C01819=1049.631,44.124,-78.703,170.591,33.560,156.310
C01820=1049.638,44.373,-78.720,170.592,33.562,156.310
C01821=1049.643,44.623,-78.737,170.594,33.564,156.311
C01822=1049.650,44.872,-78.754,170.596,33.566,156.311
C01823=1049.656,45.158,-78.774,170.597,33.568,156.311
C01824=1049.664,45.444,-78.793,170.599,33.571,156.312
C01825=1049.671,45.731,-78.812,170.601,33.573,156.312
C01826=1049.678,46.017,-78.832,170.603,33.575,156.312
C01827=1049.684,46.266,-78.848,170.605,33.577,156.313
C01828=1049.690,46.516,-78.866,170.606,33.579,156.313
C01829=1049.696,46.765,-78.883,170.608,33.581,156.313
C01830=1049.702,47.014,-78.900,170.610,33.583,156.314
C01831=1049.709,47.263,-78.917,170.611,33.585,156.314
C01832=1049.714,47.513,-78.934,170.613,33.587,156.314
C01833=1049.721,47.762,-78.951,170.615,33.589,156.315
C01834=1049.727,48.012,-78.967,170.617,33.590,156.315
C01835=1049.732,48.261,-78.985,170.619,33.592,156.315
C01836=1049.739,48.510,-79.002,170.620,33.594,156.316
C01837=1049.745,48.759,-79.018,170.622,33.596,156.316
C01838=1049.751,49.008,-79.036,170.624,33.598,156.316
C01839=1049.757,49.258,-79.053,170.625,33.600,156.316
C01840=1049.763,49.507,-79.070,170.627,33.602,156.317
C01841=1049.770,49.757,-79.088,170.629,33.604,156.317
C01842=1049.775,50.006,-79.104,170.630,33.606,156.317
C01843=1049.781,50.255,-79.121,170.632,33.608,156.318
C01844=1049.788,50.505,-79.139,170.634,33.610,156.318
C01845=1049.794,50.754,-79.155,170.635,33.612,156.318
C01846=1049.800,51.004,-79.173,170.637,33.614,156.319
C01847=1049.806,51.253,-79.190,170.638,33.616,156.319
C01848=1049.813,51.503,-79.207,170.640,33.618,156.319
C01849=1049.818,51.752,-79.224,170.642,33.620,156.320
C01850=1049.825,52.001,-79.241,170.643,33.622,156.320
C01851=1049.831,52.250,-79.258,170.645,33.624,156.320
C01852=1049.837,52.499,-79.275,170.647,33.626,156.321
C01853=1049.843,52.749,-79.293,170.648,33.628,156.321
C01854=1049.850,52.998,-79.310,170.650,33.630,156.321
C01855=1049.856,53.247,-79.327,170.652,33.632,156.322
C01856=1049.862,53.497,-79.344,170.653,33.633,156.322
C01857=1049.868,53.746,-79.362,170.655,33.635,156.322
C01858=1049.874,53.995,-79.379,170.656,33.637,156.322
C01859=1049.881,54.245,-79.396,170.658,33.639,156.323
C01860=1049.886,54.494,-79.413,170.660,33.641,156.323
C01861=1049.893,54.744,-79.430,170.661,33.643,156.323
C01862=1049.899,54.992,-79.447,170.663,33.645,156.324
C01863=1049.905,55.242,-79.465,170.665,33.647,156.324
C01864=1049.912,55.491,-79.482,170.666,33.649,156.324
C01865=1049.918,55.741,-79.499,170.668,33.651,156.325
C01866=1049.924,55.990,-79.516,170.670,33.653,156.325
C01867=1049.931,56.239,-79.534,170.671,33.655,156.325
C01868=1049.936,56.488,-79.551,170.673,33.657,156.326
C01869=1049.943,56.738,-79.568,170.674,33.659,156.326
C01870=1049.949,56.988,-79.586,170.676,33.660,156.326
C01871=1049.955,57.236,-79.603,170.678,33.662,156.326
C01872=1049.962,57.486,-79.620,170.679,33.664,156.327
C01873=1049.967,57.735,-79.638,170.681,33.666,156.327
C01874=1049.974,57.985,-79.655,170.684,33.668,156.327
C01875=1049.980,58.234,-79.672,170.685,33.670,156.328
C01876=1049.987,58.483,-79.690,170.687,33.672,156.328
C01877=1049.994,58.733,-79.707,170.689,33.674,156.328
C01878=1049.999,58.982,-79.725,170.690,33.676,156.329
C01879=1050.006,59.231,-79.742,170.692,33.678,156.329
C01880=1050.011,59.480,-79.760,170.693,33.680,156.329
C01881=1050.018,59.730,-79.777,170.695,33.682,156.330
C01882=1050.024,59.979,-79.795,170.697,33.683,156.330
C01883=1050.031,60.228,-79.812,170.698,33.685,156.330
C01884=1050.038,60.478,-79.829,170.700,33.687,156.330
C01885=1050.043,60.727,-79.847,170.702,33.689,156.331
C01886=1050.050,60.976,-79.864,170.703,33.691,156.331
C01887=1050.057,61.262,-79.884,170.705,33.693,156.331
C01888=1050.064,61.548,-79.904,170.707,33.696,156.332
C01889=1050.071,61.834,-79.924,170.709,33.698,156.332
C01890=1050.079,62.120,-79.943,170.711,33.700,156.332
C01891=1050.085,62.369,-79.961,170.712,33.702,156.333
C01892=1050.091,62.619,-79.979,170.714,33.704,156.333
C01893=1050.097,62.868,-79.996,170.716,33.706,156.333
C01894=1050.104,63.117,-80.014,170.717,33.708,156.334
C01895=1050.110,63.366,-80.032,170.719,33.710,156.334
C01896=1050.117,63.615,-80.049,170.721,33.712,156.334
C01897=1050.123,63.865,-80.067,170.722,33.713,156.335
C01898=1050.130,64.114,-80.084,170.724,33.715,156.335
C01899=1050.135,64.363,-80.102,170.726,33.717,156.335
C01900=1050.142,64.613,-80.119,170.727,33.719,156.336
C01901=1050.148,64.862,-80.137,170.729,33.721,156.336
C01902=1050.154,65.111,-80.155,170.730,33.723,156.336
C01903=1050.160,65.361,-80.173,170.732,33.725,156.337
C01904=1050.167,65.610,-80.191,170.734,33.727,156.337
C01905=1050.172,65.859,-80.208,170.735,33.729,156.337
C01906=1050.178,66.109,-80.226,170.737,33.731,156.337
C01907=1050.185,66.358,-80.244,170.739,33.733,156.338
C01908=1050.191,66.607,-80.261,170.741,33.734,156.338
C01909=1050.197,66.856,-80.280,170.743,33.736,156.338
C01910=1050.204,67.106,-80.297,170.744,33.738,156.339
C01911=1050.210,67.355,-80.315,170.746,33.741,156.339
C01912=1050.216,67.605,-80.333,170.748,33.743,156.340
C01913=1050.222,67.854,-80.351,170.749,33.745,156.340
C01914=1050.228,68.102,-80.368,170.751,33.747,156.340
C01915=1050.235,68.352,-80.386,170.753,33.749,156.340
C01916=1050.241,68.602,-80.404,170.754,33.751,156.341
C01917=1050.247,68.850,-80.422,170.756,33.753,156.341
C01918=1050.253,69.100,-80.440,170.757,33.755,156.341
C01919=1050.259,69.350,-80.458,170.759,33.757,156.342
C01920=1050.265,69.599,-80.475,170.761,33.759,156.342
C01921=1050.271,69.848,-80.494,170.762,33.761,156.342
C01922=1050.278,70.097,-80.512,170.764,33.763,156.343
C01923=1050.283,70.346,-80.529,170.766,33.764,156.343
C01924=1050.290,70.596,-80.548,170.767,33.766,156.343
C01925=1050.296,70.845,-80.565,170.769,33.768,156.344
C01926=1050.302,71.094,-80.583,170.770,33.770,156.344
C01927=1050.308,71.343,-80.602,170.772,33.772,156.344
C01928=1050.314,71.593,-80.620,170.774,33.774,156.345
C01929=1050.321,71.843,-80.638,170.775,33.776,156.345
C01930=1050.326,72.091,-80.656,170.777,33.778,156.345
C01931=1050.332,72.341,-80.674,170.779,33.780,156.346
C01932=1050.339,72.590,-80.692,170.780,33.783,156.346
C01933=1050.345,72.840,-80.710,170.782,33.785,156.346
C01934=1050.351,73.088,-80.727,170.783,33.787,156.347
C01935=1050.358,73.338,-80.746,170.786,33.789,156.347
C01936=1050.364,73.587,-80.764,170.788,33.791,156.347
C01937=1050.370,73.836,-80.782,170.789,33.792,156.348
C01938=1050.376,74.085,-80.800,170.791,33.794,156.348
C01939=1050.382,74.335,-80.819,170.792,33.796,156.348
C01940=1050.388,74.584,-80.837,170.794,33.798,156.349
C01941=1050.395,74.833,-80.855,170.796,33.800,156.349
C01942=1050.400,75.082,-80.873,170.797,33.802,156.349
C01943=1050.407,75.332,-80.892,170.799,33.804,156.350
C01944=1050.413,75.581,-80.909,170.801,33.806,156.350
C01945=1050.419,75.830,-80.928,170.802,33.808,156.350
C01946=1050.425,76.079,-80.946,170.804,33.810,156.351
C01947=1050.431,76.329,-80.964,170.805,33.812,156.351
C01948=1050.437,76.578,-80.982,170.807,33.814,156.351
C01949=1050.444,76.827,-81.000,170.809,33.816,156.352
C01950=1050.451,77.077,-81.018,170.810,33.819,156.352
C01951=1050.457,77.363,-81.040,170.812,33.821,156.352
C01952=1050.464,77.648,-81.060,170.814,33.823,156.353
C01953=1050.471,77.933,-81.081,170.816,33.825,156.353
C01954=1050.479,78.219,-81.102,170.818,33.828,156.353
C01955=1050.484,78.468,-81.120,170.819,33.830,156.354
C01956=1050.491,78.718,-81.139,170.821,33.832,156.354
C01957=1050.496,78.967,-81.158,170.823,33.834,156.354
C01958=1050.503,79.217,-81.176,170.824,33.835,156.355
C01959=1050.509,79.466,-81.195,170.827,33.837,156.355
C01960=1050.515,79.714,-81.213,170.828,33.839,156.355
C01961=1050.521,79.964,-81.231,170.830,33.842,156.356
C01962=1050.527,80.213,-81.249,170.832,33.844,156.356
C01963=1050.533,80.463,-81.269,170.833,33.846,156.357
C01964=1050.539,80.712,-81.287,170.835,33.848,156.357
C01965=1050.545,80.961,-81.305,170.837,33.850,156.357
C01966=1050.551,81.210,-81.323,170.838,33.852,156.357
C01967=1050.558,81.460,-81.341,170.840,33.854,156.358
C01968=1050.563,81.709,-81.361,170.841,33.856,156.358
C01969=1050.570,81.958,-81.379,170.843,33.858,156.359
C01970=1050.576,82.207,-81.398,170.845,33.860,156.359
C01971=1050.582,82.456,-81.416,170.846,33.862,156.359
C01972=1050.588,82.705,-81.434,170.848,33.864,156.360
C01973=1050.594,82.955,-81.453,170.849,33.866,156.360
C01974=1050.600,83.204,-81.472,170.851,33.868,156.360
C01975=1050.606,83.454,-81.490,170.853,33.871,156.361
C01976=1050.613,83.703,-81.509,170.854,33.872,156.361
C01977=1050.618,83.952,-81.528,170.856,33.874,156.361
C01978=1050.624,84.201,-81.546,170.858,33.876,156.362
C01979=1050.630,84.450,-81.564,170.859,33.878,156.362
C01980=1050.637,84.700,-81.583,170.861,33.880,156.362
C01981=1050.643,84.949,-81.601,170.863,33.882,156.363
C01982=1050.649,85.198,-81.621,170.865,33.884,156.363
C01983=1050.655,85.447,-81.639,170.867,33.887,156.363
C01984=1050.662,85.696,-81.658,170.868,33.889,156.364
C01985=1050.668,85.946,-81.676,170.870,33.891,156.364
C01986=1050.674,86.196,-81.695,170.872,33.893,156.364
C01987=1050.680,86.445,-81.714,170.873,33.895,156.365
C01988=1050.686,86.693,-81.732,170.875,33.896,156.365
C01989=1050.692,86.942,-81.751,170.876,33.898,156.365
C01990=1050.699,87.191,-81.769,170.878,33.900,156.366
C01991=1050.704,87.441,-81.789,170.880,33.902,156.366
C01992=1050.711,87.690,-81.807,170.881,33.905,156.366
C01993=1050.717,87.940,-81.825,170.883,33.907,156.367
C01994=1050.723,88.189,-81.844,170.885,33.909,156.367
C01995=1050.729,88.438,-81.863,170.886,33.911,156.367
C01996=1050.735,88.687,-81.882,170.888,33.913,156.368
C01997=1050.742,88.936,-81.900,170.890,33.915,156.368
C01998=1050.748,89.186,-81.919,170.891,33.917,156.368
C01999=1050.754,89.435,-81.938,170.893,33.919,156.369
C02000=1050.760,89.684,-81.957,170.894,33.920,156.369
C02001=1050.767,89.933,-81.976,170.896,33.922,156.369
C02002=1050.772,90.183,-81.995,170.898,33.924,156.370
C02003=1050.779,90.432,-82.013,170.900,33.926,156.370
C02004=1050.785,90.681,-82.032,170.902,33.929,156.370
C02005=1050.791,90.930,-82.051,170.904,33.931,156.371
C02006=1050.797,91.179,-82.070,170.905,33.933,156.371
C02007=1050.803,91.429,-82.089,170.907,33.935,156.371
C02008=1050.810,91.678,-82.108,170.908,33.937,156.372
C02009=1050.815,91.927,-82.127,170.910,33.939,156.372
C02010=1050.822,92.177,-82.146,170.912,33.941,156.372
C02011=1050.827,92.426,-82.165,170.913,33.943,156.373
C02012=1050.834,92.675,-82.184,170.915,33.945,156.373
C02013=1050.840,92.924,-82.204,170.917,33.948,156.374
C02014=1050.846,93.173,-82.222,170.918,33.950,156.374
C02015=1050.853,93.459,-82.244,170.920,33.952,156.374
C02016=1050.860,93.744,-82.266,170.922,33.954,156.375
C02017=1050.867,94.030,-82.287,170.924,33.957,156.375
C02018=1050.874,94.315,-82.309,170.926,33.959,156.375
C02019=1050.879,94.564,-82.328,170.927,33.961,156.376
C02020=1050.886,94.814,-82.347,170.929,33.963,156.376
C02021=1050.891,95.063,-82.366,170.932,33.965,156.376
C02022=1050.897,95.312,-82.386,170.933,33.967,156.377
C02023=1050.904,95.562,-82.405,170.935,33.969,156.377
C02024=1050.910,95.811,-82.424,170.937,33.972,156.378
C02025=1050.916,96.060,-82.443,170.938,33.973,156.378
C02026=1050.922,96.310,-82.462,170.940,33.975,156.378
C02027=1050.929,96.558,-82.482,170.941,33.977,156.379
C02028=1050.935,96.808,-82.501,170.943,33.979,156.379
C02029=1050.941,97.057,-82.520,170.945,33.981,156.379
C02030=1050.947,97.306,-82.539,170.946,33.984,156.380
C02031=1050.953,97.555,-82.558,170.948,33.986,156.380
C02032=1050.959,97.804,-82.577,170.950,33.988,156.380
C02033=1050.965,98.053,-82.597,170.951,33.990,156.381
C02034=1050.971,98.303,-82.615,170.953,33.992,156.381
C02035=1050.977,98.552,-82.635,170.955,33.994,156.381
C02036=1050.984,98.801,-82.654,170.956,33.996,156.382
C02037=1050.989,99.050,-82.673,170.958,33.998,156.382
C02038=1050.996,99.300,-82.692,170.960,34.000,156.382
C02039=1051.002,99.549,-82.712,170.962,34.002,156.383
C02040=1051.009,99.798,-82.731,170.964,34.004,156.383
C02041=1051.014,100.047,-82.750,170.966,34.006,156.383
C02042=1051.020,100.296,-82.770,170.967,34.008,156.384
C02043=1051.027,100.545,-82.789,170.969,34.010,156.384
C02044=1051.033,100.795,-82.808,170.970,34.012,156.384
C02045=1051.039,101.043,-82.828,170.972,34.014,156.385
C02046=1051.045,101.292,-82.847,170.974,34.016,156.385
C02047=1051.051,101.542,-82.866,170.975,34.019,156.386
C02048=1051.057,101.791,-82.886,170.977,34.021,156.386
C02049=1051.063,102.041,-82.905,170.979,34.023,156.386
C02050=1051.069,102.290,-82.925,170.980,34.024,156.387
C02051=1051.075,102.539,-82.944,170.982,34.027,156.387
C02052=1051.081,102.788,-82.964,170.984,34.029,156.387
C02053=1051.087,103.037,-82.983,170.985,34.031,156.388
C02054=1051.093,103.286,-83.003,170.987,34.033,156.388
C02055=1051.099,103.535,-83.022,170.989,34.035,156.388
C02056=1051.105,103.784,-83.042,170.991,34.037,156.389
C02057=1051.111,104.033,-83.061,170.993,34.039,156.389
C02058=1051.117,104.283,-83.081,170.995,34.042,156.389
C02059=1051.123,104.532,-83.101,170.996,34.044,156.390
C02060=1051.129,104.782,-83.120,170.998,34.046,156.390
C02061=1051.135,105.030,-83.140,170.999,34.048,156.390
C02062=1051.142,105.279,-83.159,171.001,34.050,156.391
C02063=1051.148,105.528,-83.178,171.003,34.052,156.391
C02064=1051.154,105.777,-83.198,171.004,34.054,156.392
C02065=1051.160,106.027,-83.218,171.006,34.056,156.392
C02066=1051.166,106.276,-83.238,171.008,34.059,156.392
C02067=1051.172,106.526,-83.257,171.009,34.060,156.393
C02068=1051.178,106.774,-83.276,171.011,34.062,156.393
C02069=1051.184,107.023,-83.296,171.013,34.064,156.393
C02070=1051.191,107.273,-83.316,171.014,34.066,156.394
C02071=1051.197,107.522,-83.336,171.016,34.069,156.394
C02072=1051.202,107.771,-83.355,171.019,34.071,156.394
C02073=1051.208,108.020,-83.375,171.020,34.073,156.395
C02074=1051.215,108.269,-83.394,171.022,34.075,156.395
C02075=1051.221,108.519,-83.414,171.024,34.077,156.396
C02076=1051.227,108.767,-83.434,171.025,34.079,156.396
C02077=1051.233,109.017,-83.453,171.027,34.081,156.396
C02078=1051.239,109.266,-83.473,171.029,34.083,156.397
C02079=1051.246,109.551,-83.496,171.031,34.086,156.397
C02080=1051.253,109.837,-83.519,171.033,34.088,156.397
C02081=1051.260,110.123,-83.541,171.035,34.090,156.398
C02082=1051.267,110.408,-83.564,171.036,34.093,156.398
C02083=1051.274,110.658,-83.583,171.038,34.095,156.399
C02084=1051.280,110.906,-83.603,171.040,34.097,156.399
C02085=1051.286,111.155,-83.623,171.041,34.099,156.399
C02086=1051.292,111.405,-83.642,171.043,34.101,156.400
C02087=1051.298,111.654,-83.663,171.045,34.103,156.400
C02088=1051.304,111.903,-83.683,171.048,34.105,156.400
C02089=1051.310,112.152,-83.703,171.049,34.107,156.401
C02090=1051.316,112.401,-83.722,171.051,34.109,156.401
C02091=1051.322,112.651,-83.742,171.053,34.111,156.401
C02092=1051.328,112.900,-83.762,171.054,34.114,156.402
C02093=1051.334,113.148,-83.782,171.056,34.116,156.402
C02094=1051.340,113.397,-83.802,171.058,34.118,156.402
C02095=1051.347,113.647,-83.822,171.059,34.120,156.403
C02096=1051.353,113.896,-83.842,171.061,34.122,156.403
C02097=1051.358,114.145,-83.862,171.063,34.124,156.404
C02098=1051.364,114.394,-83.882,171.064,34.126,156.404
C02099=1051.371,114.644,-83.903,171.066,34.129,156.404
C02100=1051.377,114.892,-83.922,171.068,34.131,156.405
C02101=1051.382,115.142,-83.943,171.069,34.133,156.405
C02102=1051.388,115.390,-83.963,171.072,34.135,156.405
C02103=1051.394,115.641,-83.983,171.074,34.137,156.406
C02104=1051.399,115.890,-84.003,171.075,34.139,156.406
C02105=1051.405,116.138,-84.023,171.077,34.141,156.407
C02106=1051.411,116.387,-84.043,171.079,34.144,156.407
C02107=1051.418,116.637,-84.063,171.080,34.146,156.407
C02108=1051.423,116.886,-84.084,171.082,34.148,156.408
C02109=1051.429,117.135,-84.104,171.084,34.150,156.408
C02110=1051.436,117.384,-84.124,171.085,34.152,156.408
C02111=1051.442,117.633,-84.144,171.087,34.154,156.409
C02112=1051.447,117.882,-84.165,171.089,34.157,156.409
C02113=1051.453,118.131,-84.185,171.090,34.159,156.410
C02114=1051.460,118.381,-84.205,171.092,34.161,156.410
C02115=1051.466,118.629,-84.225,171.094,34.163,156.410
C02116=1051.471,118.878,-84.246,171.096,34.165,156.411
C02117=1051.477,119.128,-84.266,171.098,34.168,156.411
C02118=1051.483,119.377,-84.286,171.100,34.170,156.411
C02119=1051.489,119.626,-84.306,171.102,34.172,156.412
C02120=1051.495,119.875,-84.327,171.103,34.174,156.412
C02121=1051.501,120.124,-84.347,171.105,34.176,156.413
C02122=1051.507,120.373,-84.367,171.107,34.179,156.413
C02123=1051.513,120.623,-84.388,171.108,34.180,156.413
C02124=1051.519,120.871,-84.408,171.110,34.182,156.414
C02125=1051.525,121.120,-84.428,171.112,34.185,156.414
C02126=1051.531,121.370,-84.449,171.113,34.187,156.414
C02127=1051.537,121.619,-84.469,171.115,34.189,156.415
C02128=1051.543,121.867,-84.489,171.117,34.191,156.415
C02129=1051.549,122.117,-84.510,171.119,34.193,156.416
C02130=1051.555,122.366,-84.530,171.121,34.195,156.416
C02131=1051.562,122.615,-84.550,171.123,34.198,156.416
C02132=1051.567,122.864,-84.571,171.125,34.200,156.417
C02133=1051.573,123.113,-84.591,171.126,34.202,156.417
C02134=1051.580,123.362,-84.612,171.128,34.204,156.417
C02135=1051.585,123.611,-84.632,171.130,34.206,156.418
C02136=1051.592,123.861,-84.653,171.132,34.208,156.418
C02137=1051.598,124.110,-84.673,171.133,34.211,156.419
C02138=1051.604,124.358,-84.693,171.135,34.212,156.419
C02139=1051.610,124.608,-84.714,171.137,34.214,156.419
C02140=1051.616,124.857,-84.734,171.138,34.217,156.420
C02141=1051.622,125.106,-84.754,171.140,34.219,156.420
C02142=1051.628,125.355,-84.775,171.142,34.221,156.420
C02143=1051.635,125.641,-84.799,171.145,34.223,156.421
C02144=1051.642,125.926,-84.822,171.147,34.226,156.421
C02145=1051.649,126.211,-84.846,171.149,34.228,156.422
C02146=1051.656,126.497,-84.870,171.151,34.231,156.422
C02147=1051.662,126.746,-84.890,171.153,34.233,156.422
C02148=1051.668,126.995,-84.910,171.154,34.235,156.423
C02149=1051.675,127.244,-84.932,171.156,34.237,156.423
C02150=1051.681,127.493,-84.952,171.158,34.239,156.423
C02151=1051.687,127.743,-84.972,171.160,34.241,156.424
C02152=1051.693,127.991,-84.993,171.161,34.243,156.424
C02153=1051.699,128.241,-85.013,171.163,34.246,156.425
C02154=1051.705,128.490,-85.034,171.165,34.248,156.425
C02155=1051.711,128.739,-85.055,171.167,34.250,156.425
C02156=1051.717,128.988,-85.075,171.169,34.252,156.426
C02157=1051.723,129.237,-85.096,171.171,34.254,156.426
C02158=1051.730,129.486,-85.117,171.173,34.256,156.426
C02159=1051.736,129.735,-85.137,171.175,34.259,156.427
C02160=1051.741,129.984,-85.157,171.176,34.260,156.427
C02161=1051.748,130.233,-85.179,171.178,34.262,156.427
C02162=1051.754,130.482,-85.198,171.180,34.265,156.428
C02163=1051.760,130.731,-85.220,171.182,34.267,156.428
C02164=1051.766,130.980,-85.240,171.183,34.269,156.429
C02165=1051.772,131.230,-85.261,171.185,34.271,156.429
C02166=1051.779,131.479,-85.282,171.187,34.273,156.429
C02167=1051.784,131.728,-85.303,171.189,34.275,156.430
C02168=1051.791,131.977,-85.324,171.191,34.278,156.430
C02169=1051.797,132.226,-85.344,171.193,34.280,156.430
C02170=1051.803,132.475,-85.366,171.195,34.282,156.431
C02171=1051.809,132.724,-85.386,171.197,34.284,156.431
C02172=1051.815,132.973,-85.407,171.198,34.286,156.432
C02173=1051.820,133.222,-85.428,171.200,34.289,156.432
C02174=1051.827,133.471,-85.449,171.202,34.290,156.432
C02175=1051.833,133.720,-85.470,171.204,34.293,156.433
C02176=1051.839,133.969,-85.491,171.205,34.295,156.433
C02177=1051.845,134.218,-85.512,171.207,34.297,156.434
C02178=1051.851,134.467,-85.533,171.209,34.299,156.434
C02179=1051.857,134.717,-85.554,171.211,34.301,156.434
C02180=1051.863,134.965,-85.574,171.213,34.304,156.435
C02181=1051.869,135.215,-85.596,171.215,34.306,156.435
C02182=1051.875,135.463,-85.617,171.217,34.308,156.436
C02183=1051.881,135.713,-85.638,171.219,34.310,156.436
C02184=1051.887,135.961,-85.659,171.221,34.313,156.436
C02185=1051.893,136.210,-85.681,171.222,34.315,156.437
C02186=1051.900,136.460,-85.701,171.224,34.317,156.437
C02187=1051.905,136.708,-85.722,171.226,34.319,156.437
C02188=1051.911,136.958,-85.744,171.228,34.321,156.438
C02189=1051.917,137.206,-85.764,171.229,34.324,156.438
C02190=1051.923,137.456,-85.785,171.231,34.325,156.439
C02191=1051.930,137.705,-85.807,171.233,34.328,156.439
C02192=1051.935,137.954,-85.828,171.236,34.330,156.439
C02193=1051.942,138.203,-85.849,171.238,34.332,156.440
C02194=1051.947,138.451,-85.870,171.239,34.334,156.440
C02195=1051.953,138.700,-85.891,171.241,34.336,156.440
C02196=1051.959,138.950,-85.912,171.243,34.339,156.441
C02197=1051.966,139.199,-85.933,171.245,34.341,156.441
C02198=1051.972,139.448,-85.955,171.246,34.343,156.442
C02199=1051.978,139.697,-85.976,171.248,34.345,156.442
C02200=1051.983,139.946,-85.997,171.250,34.348,156.442
C02201=1051.989,140.195,-86.019,171.252,34.350,156.443
C02202=1051.995,140.444,-86.040,171.254,34.352,156.443
C02203=1052.001,140.693,-86.061,171.256,34.354,156.444
C02204=1052.008,140.942,-86.082,171.258,34.357,156.444
C02205=1052.013,141.191,-86.103,171.260,34.359,156.444
C02206=1052.019,141.440,-86.125,171.262,34.361,156.445
C02207=1052.026,141.725,-86.150,171.264,34.364,156.445
C02208=1052.033,142.010,-86.174,171.266,34.366,156.446
C02209=1052.040,142.296,-86.198,171.268,34.369,156.446
C02210=1052.047,142.582,-86.224,171.270,34.371,156.447
C02211=1052.052,142.830,-86.245,171.272,34.373,156.447
C02212=1052.059,143.079,-86.266,171.274,34.376,156.447
C02213=1052.065,143.329,-86.287,171.276,34.378,156.448
C02214=1052.071,143.577,-86.308,171.278,34.380,156.448
C02215=1052.077,143.826,-86.330,171.280,34.382,156.448
C02216=1052.083,144.076,-86.351,171.282,34.385,156.449
C02217=1052.088,144.324,-86.373,171.284,34.387,156.449
C02218=1052.095,144.573,-86.394,171.285,34.389,156.450
C02219=1052.101,144.823,-86.416,171.287,34.392,156.450
C02220=1052.106,145.071,-86.437,171.289,34.393,156.450
C02221=1052.113,145.320,-86.459,171.291,34.396,156.451
C02222=1052.119,145.569,-86.480,171.293,34.398,156.451
C02223=1052.125,145.819,-86.502,171.295,34.400,156.452
C02224=1052.130,146.067,-86.523,171.297,34.402,156.452
C02225=1052.137,146.316,-86.545,171.299,34.405,156.453
C02226=1052.143,146.566,-86.567,171.301,34.407,156.453
C02227=1052.149,146.815,-86.588,171.303,34.409,156.453
C02228=1052.154,147.063,-86.610,171.305,34.411,156.454
C02229=1052.161,147.313,-86.631,171.307,34.414,156.454
C02230=1052.167,147.562,-86.653,171.308,34.416,156.454
C02231=1052.173,147.810,-86.675,171.310,34.418,156.455
C02232=1052.179,148.059,-86.696,171.312,34.420,156.455
C02233=1052.185,148.308,-86.718,171.314,34.423,156.456
C02234=1052.191,148.557,-86.740,171.317,34.425,156.456
C02235=1052.197,148.806,-86.761,171.319,34.427,156.456
C02236=1052.203,149.055,-86.783,171.320,34.430,156.457
C02237=1052.209,149.304,-86.804,171.322,34.432,156.457
C02238=1052.215,149.553,-86.827,171.324,34.434,156.458
C02239=1052.221,149.802,-86.849,171.326,34.436,156.458
C02240=1052.226,150.051,-86.870,171.328,34.439,156.458
C02241=1052.233,150.300,-86.892,171.330,34.440,156.459
C02242=1052.239,150.549,-86.913,171.332,34.443,156.459
C02243=1052.245,150.798,-86.936,171.333,34.445,156.460
C02244=1052.251,151.047,-86.958,171.336,34.447,156.460
C02245=1052.256,151.296,-86.979,171.338,34.450,156.460
C02246=1052.262,151.545,-87.001,171.340,34.452,156.461
C02247=1052.269,151.794,-87.022,171.342,34.454,156.461
C02248=1052.275,152.043,-87.045,171.344,34.457,156.462
C02249=1052.280,152.292,-87.067,171.345,34.459,156.462
C02250=1052.286,152.541,-87.088,171.347,34.461,156.463
C02251=1052.293,152.789,-87.111,171.349,34.463,156.463
C02252=1052.299,153.039,-87.132,171.351,34.466,156.463
C02253=1052.305,153.288,-87.154,171.353,34.468,156.464
C02254=1052.311,153.537,-87.177,171.356,34.470,156.464
C02255=1052.317,153.786,-87.199,171.358,34.473,156.465
C02256=1052.322,154.034,-87.220,171.360,34.475,156.465
C02257=1052.329,154.283,-87.242,171.361,34.477,156.465
C02258=1052.335,154.532,-87.264,171.363,34.480,156.466
C02259=1052.340,154.782,-87.286,171.365,34.482,156.466
C02260=1052.347,155.030,-87.308,171.367,34.484,156.467
C02261=1052.353,155.279,-87.330,171.369,34.487,156.467
C02262=1052.358,155.529,-87.352,171.371,34.489,156.467
C02263=1052.364,155.777,-87.374,171.373,34.491,156.468
C02264=1052.370,156.026,-87.396,171.376,34.494,156.468
C02265=1052.376,156.275,-87.419,171.377,34.495,156.469
C02266=1052.382,156.524,-87.440,171.379,34.498,156.469
C02267=1052.389,156.773,-87.463,171.381,34.501,156.470
C02268=1052.394,157.022,-87.485,171.383,34.502,156.470
C02269=1052.401,157.271,-87.507,171.385,34.505,156.470
C02270=1052.406,157.520,-87.530,171.387,34.507,156.471
C02271=1052.413,157.805,-87.555,171.389,34.510,156.471
C02272=1052.420,158.090,-87.580,171.391,34.513,156.472
C02273=1052.426,158.375,-87.605,171.394,34.515,156.472
C02274=1052.434,158.660,-87.631,171.397,34.518,156.473
C02275=1052.440,158.909,-87.653,171.399,34.520,156.473
C02276=1052.446,159.158,-87.675,171.400,34.523,156.473
C02277=1052.451,159.407,-87.697,171.402,34.525,156.474
C02278=1052.458,159.655,-87.719,171.404,34.527,156.474
C02279=1052.463,159.904,-87.742,171.406,34.530,156.475
C02280=1052.469,160.153,-87.764,171.408,34.531,156.475
C02281=1052.476,160.402,-87.786,171.411,34.534,156.475
C02282=1052.481,160.652,-87.809,171.413,34.537,156.476
C02283=1052.488,160.900,-87.831,171.415,34.538,156.476
C02284=1052.494,161.149,-87.854,171.417,34.541,156.477
C02285=1052.499,161.399,-87.876,171.419,34.543,156.477
C02286=1052.505,161.647,-87.899,171.421,34.546,156.478
C02287=1052.511,161.896,-87.921,171.422,34.548,156.478
C02288=1052.517,162.146,-87.944,171.424,34.551,156.479
C02289=1052.522,162.394,-87.967,171.426,34.554,156.479
C02290=1052.527,162.643,-87.989,171.429,34.555,156.479
C02291=1052.534,162.891,-88.012,171.431,34.558,156.480
C02292=1052.539,163.141,-88.034,171.433,34.560,156.480
C02293=1052.545,163.390,-88.057,171.435,34.563,156.481
C02294=1052.551,163.639,-88.080,171.437,34.565,156.481
C02295=1052.557,163.887,-88.102,171.439,34.568,156.482
C02296=1052.563,164.137,-88.124,171.441,34.571,156.482
C02297=1052.568,164.386,-88.147,171.442,34.573,156.483
C02298=1052.574,164.634,-88.170,171.445,34.575,156.483
C02299=1052.581,164.883,-88.192,171.447,34.577,156.483
C02300=1052.586,165.132,-88.215,171.449,34.580,156.484
C02301=1052.592,165.381,-88.238,171.451,34.582,156.484
C02302=1052.598,165.630,-88.261,171.453,34.585,156.485
C02303=1052.603,165.879,-88.284,171.455,34.587,156.485
C02304=1052.610,166.128,-88.306,171.457,34.590,156.486
C02305=1052.615,166.377,-88.329,171.459,34.592,156.486
C02306=1052.621,166.626,-88.352,171.461,34.594,156.486
C02307=1052.627,166.875,-88.375,171.464,34.597,156.487
C02308=1052.633,167.123,-88.397,171.466,34.599,156.487
C02309=1052.639,167.372,-88.420,171.468,34.602,156.488
C02310=1052.645,167.622,-88.442,171.470,34.604,156.488
C02311=1052.650,167.870,-88.465,171.472,34.607,156.489
C02312=1052.656,168.119,-88.488,171.474,34.610,156.489
C02313=1052.662,168.368,-88.511,171.476,34.611,156.489
C02314=1052.668,168.617,-88.533,171.477,34.614,156.490
C02315=1052.674,168.866,-88.556,171.480,34.616,156.490
C02316=1052.680,169.115,-88.579,171.482,34.619,156.491
C02317=1052.685,169.364,-88.602,171.484,34.621,156.491
C02318=1052.691,169.612,-88.625,171.486,34.624,156.492
C02319=1052.698,169.861,-88.648,171.488,34.626,156.492
C02320=1052.703,170.110,-88.671,171.490,34.628,156.493
C02321=1052.709,170.359,-88.693,171.492,34.631,156.493
C02322=1052.715,170.608,-88.716,171.494,34.633,156.493
C02323=1052.721,170.857,-88.739,171.497,34.636,156.494
C02324=1052.727,171.105,-88.762,171.499,34.638,156.494
C02325=1052.733,171.355,-88.785,171.501,34.641,156.495
C02326=1052.739,171.603,-88.809,171.503,34.643,156.495
C02327=1052.745,171.852,-88.832,171.505,34.646,156.496
C02328=1052.751,172.101,-88.855,171.507,34.648,156.496
C02329=1052.757,172.350,-88.878,171.509,34.650,156.497
C02330=1052.763,172.598,-88.900,171.511,34.653,156.497
C02331=1052.769,172.847,-88.923,171.514,34.655,156.497
C02332=1052.774,173.096,-88.946,171.516,34.658,156.498
C02333=1052.781,173.346,-88.969,171.518,34.660,156.498
C02334=1052.787,173.595,-88.992,171.520,34.663,156.499
C02335=1052.794,173.878,-89.018,171.523,34.665,156.499
C02336=1052.800,174.163,-89.045,171.525,34.669,156.500
C02337=1052.808,174.448,-89.071,171.527,34.671,156.500
C02338=1052.814,174.732,-89.098,171.530,34.674,156.501
C02339=1052.820,174.981,-89.121,171.532,34.676,156.501
C02340=1052.826,175.230,-89.143,171.534,34.679,156.502
C02341=1052.832,175.478,-89.167,171.537,34.681,156.502
C02342=1052.838,175.728,-89.190,171.539,34.684,156.503
C02343=1052.844,175.977,-89.213,171.541,34.686,156.503
C02344=1052.850,176.226,-89.236,171.543,34.689,156.504
C02345=1052.856,176.474,-89.260,171.546,34.691,156.504
C02346=1052.862,176.724,-89.283,171.548,34.694,156.504
C02347=1052.868,176.972,-89.306,171.550,34.696,156.505
C02348=1052.875,177.220,-89.329,171.552,34.698,156.505
C02349=1052.880,177.469,-89.352,171.554,34.701,156.506
C02350=1052.887,177.719,-89.375,171.556,34.703,156.506
C02351=1052.893,177.967,-89.399,171.558,34.706,156.507
C02352=1052.899,178.216,-89.422,171.560,34.708,156.507
C02353=1052.904,178.465,-89.445,171.563,34.711,156.508
C02354=1052.911,178.714,-89.469,171.565,34.713,156.508
C02355=1052.917,178.963,-89.492,171.567,34.716,156.508
C02356=1052.922,179.212,-89.515,171.569,34.717,156.509
C02357=1052.929,179.461,-89.539,171.571,34.720,156.509
C02358=1052.936,179.709,-89.561,171.573,34.722,156.510
C02359=1052.941,179.958,-89.584,171.575,34.725,156.510
C02360=1052.947,180.206,-89.608,171.578,34.727,156.511
C02361=1052.954,180.456,-89.631,171.581,34.730,156.511
C02362=1052.960,180.704,-89.655,171.583,34.732,156.512
C02363=1052.965,180.953,-89.678,171.585,34.735,156.512
C02364=1052.972,181.202,-89.702,171.587,34.737,156.512
C02365=1052.978,181.451,-89.725,171.589,34.740,156.513
C02366=1052.984,181.699,-89.748,171.591,34.742,156.513
C02367=1052.990,181.949,-89.771,171.593,34.744,156.514
C02368=1052.996,182.197,-89.795,171.596,34.747,156.514
C02369=1053.002,182.447,-89.818,171.598,34.749,156.515
C02370=1053.009,182.695,-89.842,171.600,34.752,156.515
C02371=1053.015,182.944,-89.864,171.603,34.754,156.516
C02372=1053.022,183.193,-89.888,171.605,34.757,156.516
C02373=1053.027,183.442,-89.911,171.607,34.759,156.516
C02374=1053.033,183.690,-89.935,171.609,34.762,156.517
C02375=1053.040,183.939,-89.958,171.612,34.764,156.517
C02376=1053.046,184.188,-89.982,171.614,34.767,156.518
C02377=1053.051,184.438,-90.006,171.616,34.769,156.518
C02378=1053.057,184.686,-90.030,171.618,34.772,156.519
C02379=1053.063,184.935,-90.054,171.620,34.774,156.519
C02380=1053.068,185.183,-90.077,171.622,34.777,156.520
C02381=1053.075,185.432,-90.101,171.625,34.780,156.520
C02382=1053.080,185.681,-90.125,171.628,34.783,156.521
C02383=1053.086,185.929,-90.149,171.630,34.785,156.521
C02384=1053.092,186.179,-90.173,171.632,34.788,156.522
C02385=1053.098,186.427,-90.196,171.634,34.791,156.522
C02386=1053.103,186.676,-90.221,171.636,34.793,156.523
C02387=1053.110,186.925,-90.245,171.638,34.796,156.523
C02388=1053.115,187.174,-90.268,171.641,34.798,156.524
C02389=1053.121,187.422,-90.292,171.643,34.801,156.524
C02390=1053.127,187.672,-90.316,171.645,34.804,156.525
C02391=1053.133,187.920,-90.340,171.648,34.806,156.525
C02392=1053.139,188.168,-90.364,171.650,34.809,156.526
C02393=1053.145,188.418,-90.388,171.652,34.811,156.526
C02394=1053.151,188.667,-90.411,171.654,34.814,156.527
C02395=1053.156,188.916,-90.436,171.657,34.817,156.527
C02396=1053.163,189.164,-90.460,171.659,34.819,156.528
C02397=1053.168,189.413,-90.484,171.661,34.822,156.528
C02398=1053.174,189.662,-90.508,171.663,34.825,156.529
C02399=1053.181,189.946,-90.535,171.666,34.827,156.529
C02400=1053.188,190.229,-90.563,171.668,34.830,156.530
C02401=1053.194,190.514,-90.591,171.672,34.834,156.530
C02402=1053.201,190.798,-90.618,171.674,34.837,156.531
C02403=1053.207,191.047,-90.642,171.676,34.839,156.531
C02404=1053.212,191.296,-90.666,171.678,34.842,156.532
C02405=1053.218,191.544,-90.690,171.681,34.845,156.532
C02406=1053.224,191.794,-90.714,171.683,34.847,156.533
C02407=1053.230,192.042,-90.738,171.686,34.850,156.533
C02408=1053.236,192.291,-90.762,171.688,34.853,156.534
C02409=1053.242,192.540,-90.786,171.690,34.855,156.534
C02410=1053.248,192.789,-90.811,171.692,34.858,156.535
C02411=1053.254,193.037,-90.834,171.695,34.860,156.535
C02412=1053.260,193.286,-90.859,171.697,34.863,156.536
C02413=1053.266,193.534,-90.883,171.700,34.866,156.536
C02414=1053.272,193.783,-90.908,171.702,34.868,156.537
C02415=1053.278,194.032,-90.932,171.704,34.871,156.537
C02416=1053.284,194.281,-90.956,171.706,34.874,156.538
C02417=1053.290,194.529,-90.980,171.709,34.876,156.538
C02418=1053.296,194.779,-91.005,171.711,34.879,156.539
C02419=1053.302,195.027,-91.028,171.714,34.882,156.539
C02420=1053.308,195.276,-91.053,171.716,34.885,156.540
C02421=1053.314,195.524,-91.076,171.718,34.887,156.540
C02422=1053.320,195.774,-91.101,171.721,34.890,156.541
C02423=1053.327,196.022,-91.126,171.723,34.893,156.541
C02424=1053.332,196.271,-91.150,171.725,34.895,156.542
C02425=1053.338,196.520,-91.175,171.728,34.898,156.542
C02426=1053.344,196.768,-91.198,171.730,34.901,156.543
C02427=1053.350,197.017,-91.223,171.733,34.903,156.543
C02428=1053.357,197.266,-91.248,171.735,34.906,156.544
C02429=1053.362,197.514,-91.272,171.737,34.909,156.544
C02430=1053.369,197.763,-91.296,171.739,34.911,156.545
C02431=1053.374,198.012,-91.320,171.743,34.914,156.545
C02432=1053.381,198.261,-91.346,171.745,34.917,156.546
C02433=1053.387,198.510,-91.370,171.747,34.919,156.546
C02434=1053.393,198.758,-91.394,171.749,34.922,156.547
C02435=1053.399,199.007,-91.418,171.752,34.925,156.547
C02436=1053.405,199.256,-91.443,171.754,34.927,156.548
C02437=1053.411,199.504,-91.467,171.757,34.930,156.548
C02438=1053.417,199.753,-91.492,171.759,34.933,156.549
C02439=1053.423,200.001,-91.517,171.761,34.935,156.549
C02440=1053.430,200.250,-91.541,171.764,34.938,156.550
C02441=1053.435,200.500,-91.565,171.766,34.941,156.550
C02442=1053.442,200.748,-91.590,171.768,34.943,156.551
C02443=1053.448,200.997,-91.614,171.772,34.946,156.551
C02444=1053.454,201.246,-91.639,171.774,34.949,156.552
C02445=1053.461,201.494,-91.664,171.776,34.952,156.552
C02446=1053.466,201.743,-91.688,171.778,34.954,156.553
C02447=1053.472,201.991,-91.713,171.781,34.957,156.553
C02448=1053.478,202.241,-91.738,171.783,34.960,156.554
C02449=1053.484,202.488,-91.762,171.786,34.963,156.554
C02450=1053.490,202.738,-91.787,171.788,34.965,156.555
C02451=1053.496,202.986,-91.812,171.791,34.968,156.555
C02452=1053.502,203.235,-91.836,171.793,34.971,156.556
C02453=1053.508,203.484,-91.862,171.795,34.974,156.556
C02454=1053.514,203.733,-91.886,171.798,34.977,156.557
C02455=1053.519,203.981,-91.911,171.801,34.979,156.557
C02456=1053.525,204.230,-91.936,171.803,34.982,156.558
C02457=1053.532,204.479,-91.961,171.805,34.985,156.558
C02458=1053.538,204.727,-91.986,171.807,34.988,156.559
C02459=1053.544,204.976,-92.010,171.810,34.991,156.560
C02460=1053.550,205.224,-92.036,171.813,34.994,156.560
C02461=1053.556,205.473,-92.061,171.815,34.997,156.561
C02462=1053.561,205.722,-92.085,171.818,34.999,156.561
C02463=1053.587,206.773,-92.191,172.030,35.092,156.577
C02464=1053.594,207.017,-92.216,172.033,35.096,156.578
C02465=1053.599,207.260,-92.242,172.034,35.100,156.578
C02466=1053.606,207.504,-92.267,172.036,35.103,156.579
C02467=1053.612,207.747,-92.293,172.038,35.106,156.580
C02468=1053.618,207.991,-92.318,172.040,35.110,156.580
C02469=1053.624,208.235,-92.344,172.042,35.113,156.581
C02470=1053.630,208.478,-92.368,172.044,35.117,156.582
C02471=1053.637,208.722,-92.394,172.045,35.121,156.582
C02472=1053.643,208.971,-92.420,172.048,35.124,156.583
C02473=1053.649,209.219,-92.446,172.050,35.128,156.584
C02474=1053.656,209.467,-92.473,172.052,35.132,156.585
C02475=1053.662,209.716,-92.499,172.054,35.135,156.585
C02476=1053.668,209.965,-92.525,172.056,35.139,156.586
C02477=1053.675,210.213,-92.550,172.058,35.142,156.587
C02478=1053.681,210.462,-92.577,172.059,35.146,156.587
C02479=1053.687,210.710,-92.603,172.062,35.150,156.588
C02480=1053.694,210.959,-92.628,172.064,35.153,156.589
C02481=1053.700,211.208,-92.655,172.065,35.157,156.590
C02482=1053.707,211.456,-92.681,172.067,35.160,156.590
C02483=1053.713,211.705,-92.707,172.070,35.164,156.591
C02484=1053.719,211.953,-92.733,172.072,35.168,156.592
C02485=1053.726,212.202,-92.760,172.073,35.171,156.593
C02486=1053.731,212.450,-92.787,172.076,35.175,156.593
C02487=1053.738,212.699,-92.812,172.078,35.179,156.594
C02488=1053.744,212.948,-92.839,172.080,35.182,156.595
C02489=1053.751,213.196,-92.865,172.081,35.186,156.595
C02490=1053.756,213.444,-92.892,172.084,35.189,156.596
C02491=1053.763,213.693,-92.918,172.086,35.193,156.597
C02492=1053.769,213.942,-92.944,172.088,35.197,156.598
C02493=1053.775,214.190,-92.970,172.090,35.200,156.598
C02494=1053.781,214.438,-92.997,172.092,35.204,156.599
C02495=1053.788,214.687,-93.023,172.094,35.207,156.600
C02496=1053.794,214.936,-93.050,172.096,35.211,156.600
C02497=1053.801,215.184,-93.076,172.098,35.215,156.601
C02498=1053.807,215.433,-93.103,172.100,35.218,156.602
C02499=1053.813,215.681,-93.129,172.102,35.222,156.603
C02500=1053.820,215.930,-93.155,172.105,35.226,156.603
C02501=1053.825,216.179,-93.182,172.106,35.229,156.604
C02502=1053.832,216.427,-93.208,172.108,35.233,156.605
C02503=1053.838,216.676,-93.235,172.110,35.236,156.605
C02504=1053.845,216.924,-93.261,172.113,35.240,156.606
C02505=1053.850,217.172,-93.288,172.114,35.244,156.607
C02506=1053.858,217.421,-93.314,172.116,35.247,156.608
C02507=1053.863,217.669,-93.341,172.119,35.251,156.608
C02508=1053.870,217.918,-93.368,172.121,35.254,156.609
C02509=1053.876,218.167,-93.394,172.123,35.258,156.610
C02510=1053.882,218.415,-93.420,172.124,35.262,156.611
C02511=1053.889,218.664,-93.447,172.127,35.265,156.611
C02512=1053.895,218.912,-93.473,172.129,35.268,156.612
C02513=1053.902,219.161,-93.500,172.131,35.272,156.613
C02514=1053.908,219.409,-93.526,172.134,35.276,156.613
C02515=1053.914,219.658,-93.553,172.135,35.279,156.614
C02516=1053.921,219.906,-93.580,172.137,35.283,156.615
C02517=1053.927,220.155,-93.607,172.139,35.286,156.615
C02518=1053.934,220.403,-93.633,172.142,35.290,156.616
C02519=1053.940,220.652,-93.660,172.144,35.294,156.617
C02520=1053.946,220.898,-93.686,172.146,35.297,156.618
C02521=1053.952,221.144,-93.713,172.148,35.300,156.618
C02522=1053.959,221.391,-93.740,172.150,35.304,156.619
C02523=1053.964,221.637,-93.766,172.152,35.307,156.620
C02524=1053.971,221.883,-93.793,172.154,35.311,156.620
C02525=1053.977,222.129,-93.819,172.157,35.315,156.621
C02526=1053.984,222.375,-93.847,172.158,35.318,156.622
C02527=1053.989,222.621,-93.873,172.160,35.322,156.623
C02528=1053.996,222.870,-93.900,172.163,35.325,156.623
C02529=1054.002,223.118,-93.926,172.165,35.329,156.624
C02530=1054.009,223.367,-93.953,172.167,35.333,156.625
C02531=1054.014,223.615,-93.980,172.168,35.336,156.625
C02532=1054.021,223.864,-94.007,172.171,35.340,156.626
C02533=1054.027,224.112,-94.034,172.173,35.343,156.627
C02534=1054.033,224.361,-94.061,172.175,35.346,156.628
C02535=1054.039,224.610,-94.088,172.178,35.350,156.628
C02536=1054.047,224.858,-94.115,172.180,35.354,156.629
C02537=1054.052,225.106,-94.142,172.182,35.357,156.630
C02538=1054.059,225.355,-94.169,172.184,35.361,156.630
C02539=1054.065,225.603,-94.196,172.186,35.364,156.631
C02540=1054.071,225.852,-94.223,172.188,35.368,156.632
C02541=1054.077,226.100,-94.251,172.190,35.372,156.633
C02542=1054.084,226.349,-94.278,172.193,35.375,156.633
C02543=1054.091,226.597,-94.304,172.195,35.379,156.634
C02544=1054.097,226.845,-94.331,172.197,35.382,156.635
C02545=1054.103,227.094,-94.358,172.200,35.385,156.635
C02546=1054.109,227.342,-94.386,172.201,35.389,156.636
C02547=1054.116,227.591,-94.413,172.203,35.393,156.637
C02548=1054.121,227.839,-94.439,172.206,35.396,156.638
C02549=1054.128,228.088,-94.467,172.208,35.400,156.638
C02550=1054.134,228.337,-94.494,172.210,35.403,156.639
C02551=1054.141,228.584,-94.521,172.212,35.406,156.640
C02552=1054.148,228.833,-94.548,172.215,35.410,156.640
C02553=1054.154,229.082,-94.576,172.217,35.414,156.641
C02554=1054.160,229.330,-94.602,172.219,35.417,156.642
C02555=1054.167,229.579,-94.630,172.222,35.421,156.642
C02556=1054.173,229.826,-94.657,172.224,35.424,156.643
C02557=1054.179,230.075,-94.684,172.225,35.428,156.644
C02558=1054.185,230.324,-94.713,172.228,35.432,156.645
C02559=1054.191,230.573,-94.739,172.230,35.435,156.645
C02560=1054.198,230.821,-94.767,172.232,35.438,156.646
C02561=1054.204,231.069,-94.795,172.234,35.442,156.647
C02562=1054.210,231.318,-94.822,172.237,35.445,156.647
C02563=1054.217,231.566,-94.849,172.239,35.449,156.648
C02564=1054.223,231.814,-94.877,172.241,35.453,156.649
C02565=1054.229,232.063,-94.904,172.244,35.456,156.650
C02566=1054.236,232.311,-94.931,172.246,35.460,156.650
C02567=1054.242,232.559,-94.959,172.248,35.463,156.651
C02568=1054.248,232.809,-94.986,172.251,35.466,156.652
C02569=1054.254,233.057,-95.014,172.253,35.470,156.652
C02570=1054.260,233.305,-95.041,172.254,35.474,156.653
C02571=1054.267,233.553,-95.069,172.257,35.477,156.654
C02572=1054.273,233.802,-95.097,172.259,35.481,156.655
C02573=1054.279,234.050,-95.124,172.261,35.484,156.655
C02574=1054.285,234.299,-95.152,172.264,35.488,156.656
C02575=1054.292,234.547,-95.180,172.266,35.492,156.657
C02576=1054.298,234.790,-95.206,172.268,35.495,156.657
C02577=1054.304,235.032,-95.233,172.270,35.498,156.658
C02578=1054.310,235.274,-95.260,172.273,35.502,156.659
C02579=1054.316,235.517,-95.287,172.275,35.505,156.660
C02580=1054.322,235.759,-95.314,172.277,35.508,156.660
C02581=1054.328,236.001,-95.342,172.280,35.512,156.661
C02582=1054.334,236.243,-95.369,172.282,35.516,156.662
C02583=1054.340,236.486,-95.396,172.284,35.519,156.662
C02584=1054.347,236.734,-95.423,172.287,35.522,156.663
C02585=1054.354,236.983,-95.451,172.289,35.526,156.664
C02586=1054.360,237.231,-95.479,172.291,35.529,156.664
C02587=1054.366,237.479,-95.507,172.294,35.533,156.665
C02588=1054.372,237.728,-95.535,172.296,35.536,156.666
C02589=1054.379,237.976,-95.562,172.298,35.540,156.667
C02590=1054.385,238.225,-95.591,172.300,35.543,156.667
C02591=1054.391,238.473,-95.618,172.303,35.547,156.668
C02592=1054.398,238.721,-95.646,172.305,35.550,156.669
C02593=1054.405,238.969,-95.673,172.307,35.554,156.669
C02594=1054.410,239.218,-95.702,172.310,35.557,156.670
C02595=1054.417,239.467,-95.730,172.312,35.561,156.671
C02596=1054.422,239.715,-95.758,172.314,35.565,156.672
C02597=1054.429,239.963,-95.785,172.317,35.568,156.672
C02598=1054.436,240.212,-95.813,172.319,35.571,156.673
C02599=1054.442,240.460,-95.841,172.321,35.575,156.674
C02600=1054.448,240.709,-95.869,172.324,35.578,156.674
C02601=1054.455,240.957,-95.897,172.326,35.582,156.675
C02602=1054.460,241.205,-95.925,172.328,35.585,156.676
C02603=1054.467,241.453,-95.953,172.331,35.588,156.676
C02604=1054.474,241.702,-95.981,172.333,35.592,156.677
C02605=1054.480,241.950,-96.009,172.335,35.596,156.678
C02606=1054.487,242.199,-96.037,172.338,35.599,156.679
C02607=1054.493,242.447,-96.065,172.340,35.603,156.679
C02608=1054.498,242.696,-96.093,172.342,35.606,156.680
C02609=1054.505,242.943,-96.122,172.345,35.610,156.681
C02610=1054.511,243.192,-96.150,172.347,35.613,156.681
C02611=1054.518,243.441,-96.178,172.349,35.616,156.682
C02612=1054.524,243.689,-96.207,172.352,35.620,156.683
C02613=1054.531,243.937,-96.235,172.354,35.624,156.684
C02614=1054.537,244.186,-96.263,172.356,35.627,156.684
C02615=1054.542,244.434,-96.291,172.359,35.631,156.685
C02616=1054.549,244.682,-96.319,172.361,35.634,156.686
C02617=1054.555,244.930,-96.348,172.363,35.638,156.687
C02618=1054.562,245.178,-96.376,172.367,35.641,156.687
C02619=1054.568,245.427,-96.404,172.369,35.645,156.688
C02620=1054.574,245.676,-96.433,172.371,35.648,156.689
C02621=1054.581,245.924,-96.461,172.374,35.652,156.689
C02622=1054.587,246.172,-96.489,172.376,35.655,156.690
C02623=1054.593,246.421,-96.518,172.378,35.659,156.691
C02624=1054.598,246.669,-96.546,172.381,35.662,156.692
C02625=1054.605,246.917,-96.574,172.383,35.666,156.692
C02626=1054.611,247.165,-96.603,172.385,35.670,156.693
C02627=1054.617,247.414,-96.632,172.388,35.673,156.694
C02628=1054.623,247.662,-96.661,172.390,35.677,156.695
C02629=1054.629,247.911,-96.689,172.392,35.680,156.695
C02630=1054.636,248.159,-96.717,172.396,35.684,156.696
C02631=1054.643,248.407,-96.746,172.398,35.687,156.697
C02632=1054.648,248.646,-96.774,172.400,35.690,156.697
C02633=1054.654,248.886,-96.801,172.403,35.694,156.698
C02634=1054.660,249.125,-96.829,172.405,35.698,156.699
C02635=1054.666,249.365,-96.857,172.407,35.701,156.700
C02636=1054.672,249.603,-96.884,172.410,35.704,156.700
C02637=1054.678,249.843,-96.912,172.412,35.708,156.701
C02638=1054.684,250.082,-96.939,172.414,35.711,156.702
C02639=1054.690,250.321,-96.967,172.417,35.714,156.702
C02640=1054.696,250.570,-96.995,172.419,35.718,156.703
C02641=1054.702,250.818,-97.024,172.421,35.721,156.704
C02642=1054.708,251.066,-97.054,172.424,35.725,156.705
C02643=1054.715,251.314,-97.082,172.426,35.728,156.705
C02644=1054.721,251.563,-97.110,172.429,35.732,156.706
C02645=1054.727,251.811,-97.139,172.432,35.736,156.707
C02646=1054.734,252.059,-97.168,172.434,35.739,156.707
C02647=1054.740,252.308,-97.197,172.436,35.743,156.708
C02648=1054.746,252.556,-97.226,172.439,35.746,156.709
C02649=1054.752,252.804,-97.255,172.441,35.749,156.710
C02650=1054.758,253.052,-97.284,172.443,35.753,156.710
C02651=1054.765,253.301,-97.312,172.447,35.756,156.711
C02652=1054.771,253.549,-97.341,172.449,35.760,156.712
C02653=1054.777,253.797,-97.370,172.451,35.764,156.712
C02654=1054.784,254.045,-97.399,172.454,35.767,156.713
C02655=1054.790,254.293,-97.428,172.456,35.771,156.714
C02656=1054.797,254.542,-97.457,172.459,35.774,156.715
C02657=1054.803,254.791,-97.485,172.462,35.777,156.715
C02658=1054.809,255.039,-97.514,172.464,35.781,156.716
C02659=1054.815,255.287,-97.544,172.467,35.784,156.717
C02660=1054.821,255.535,-97.573,172.469,35.788,156.718
C02661=1054.828,255.783,-97.601,172.471,35.791,156.718
C02662=1054.835,256.031,-97.630,172.475,35.795,156.719
C02663=1054.841,256.279,-97.659,172.477,35.799,156.720
C02664=1054.847,256.528,-97.688,172.479,35.802,156.720
C02665=1054.854,256.776,-97.718,172.482,35.805,156.721
C02666=1054.860,257.025,-97.747,172.484,35.809,156.722
C02667=1054.867,257.273,-97.776,172.487,35.812,156.723
C02668=1054.873,257.521,-97.805,172.490,35.816,156.723
C02669=1054.879,257.769,-97.834,172.492,35.819,156.724
C02670=1054.885,258.017,-97.863,172.494,35.822,156.725
C02671=1054.892,258.266,-97.892,172.498,35.826,156.725
C02672=1054.898,258.514,-97.921,172.500,35.829,156.726
C02673=1054.905,258.762,-97.950,172.502,35.833,156.727
C02674=1054.911,259.010,-97.979,172.505,35.837,156.728
C02675=1054.917,259.258,-98.008,172.507,35.840,156.728
C02676=1054.924,259.507,-98.038,172.511,35.843,156.729
C02677=1054.931,259.755,-98.066,172.513,35.847,156.730
C02678=1054.937,260.003,-98.095,172.515,35.850,156.730
C02679=1054.944,260.251,-98.124,172.519,35.854,156.731
C02680=1054.951,260.500,-98.154,172.521,35.857,156.732
C02681=1054.957,260.748,-98.183,172.523,35.861,156.733
C02682=1054.963,260.996,-98.212,172.526,35.864,156.733
C02683=1054.969,261.244,-98.241,172.529,35.867,156.734
C02684=1054.976,261.493,-98.271,172.531,35.871,156.735
C02685=1054.983,261.741,-98.300,172.534,35.874,156.736
C02686=1054.989,261.988,-98.330,172.536,35.878,156.736
C02687=1054.996,262.237,-98.359,172.539,35.881,156.737
C02688=1055.001,262.476,-98.387,172.542,35.885,156.738
C02689=1055.008,262.714,-98.415,172.544,35.888,156.738
C02690=1055.015,262.953,-98.443,172.546,35.891,156.739
C02691=1055.021,263.191,-98.472,172.550,35.895,156.740
C02692=1055.026,263.429,-98.500,172.552,35.898,156.740
C02693=1055.032,263.668,-98.529,172.555,35.901,156.741
C02694=1055.039,263.906,-98.557,172.557,35.905,156.742
C02695=1055.044,264.144,-98.585,172.559,35.908,156.743
C02696=1055.051,264.392,-98.615,172.563,35.912,156.743
C02697=1055.057,264.641,-98.645,172.565,35.915,156.744
C02698=1055.063,264.888,-98.675,172.567,35.919,156.745
C02699=1055.070,265.137,-98.704,172.570,35.922,156.746
C02700=1055.076,265.386,-98.734,172.573,35.925,156.746
C02701=1055.082,265.633,-98.764,172.575,35.929,156.747
C02702=1055.088,265.881,-98.793,172.578,35.932,156.748
C02703=1055.095,266.130,-98.823,172.581,35.936,156.748
C02704=1055.101,266.378,-98.852,172.584,35.940,156.749
C02705=1055.108,266.625,-98.882,172.586,35.943,156.750
C02706=1055.114,266.875,-98.912,172.589,35.947,156.751
C02707=1055.120,267.122,-98.942,172.592,35.950,156.751
C02708=1055.127,267.370,-98.972,172.594,35.954,156.752
C02709=1055.133,267.619,-99.002,172.598,35.957,156.753
C02710=1055.140,267.866,-99.031,172.600,35.961,156.754
C02711=1055.146,268.114,-99.060,172.602,35.964,156.754
C02712=1055.152,268.363,-99.091,172.606,35.968,156.755
C02713=1055.159,268.610,-99.121,172.608,35.971,156.756
C02714=1055.165,268.860,-99.151,172.610,35.975,156.757
C02715=1055.171,269.107,-99.181,172.614,35.979,156.757
C02716=1055.177,269.355,-99.211,172.616,35.982,156.758
C02717=1055.184,269.604,-99.240,172.619,35.986,156.759
C02718=1055.190,269.852,-99.271,172.622,35.989,156.760
C02719=1055.196,270.099,-99.300,172.624,35.993,156.760
C02720=1055.203,270.348,-99.330,172.627,35.996,156.761
C02721=1055.209,270.596,-99.360,172.630,36.000,156.762
C02722=1055.216,270.844,-99.391,172.633,36.003,156.763
C02723=1055.222,271.092,-99.421,172.635,36.007,156.763
C02724=1055.228,271.340,-99.450,172.638,36.010,156.764
C02725=1055.235,271.588,-99.480,172.641,36.014,156.765
C02726=1055.241,271.836,-99.511,172.644,36.017,156.766
C02727=1055.248,272.084,-99.541,172.646,36.021,156.766
C02728=1055.254,272.332,-99.571,172.649,36.024,156.767
C02729=1055.261,272.580,-99.601,172.652,36.028,156.768
C02730=1055.266,272.829,-99.631,172.655,36.032,156.769
C02731=1055.273,273.077,-99.662,172.658,36.035,156.769
C02732=1055.279,273.325,-99.692,172.660,36.039,156.770
C02733=1055.285,273.573,-99.722,172.663,36.042,156.771
C02734=1055.291,273.821,-99.753,172.666,36.046,156.772
C02735=1055.298,274.069,-99.782,172.669,36.049,156.772
C02736=1055.304,274.317,-99.813,172.672,36.053,156.773
C02737=1055.310,274.565,-99.843,172.674,36.056,156.774
C02738=1055.317,274.813,-99.874,172.677,36.060,156.775
C02739=1055.323,275.061,-99.904,172.680,36.063,156.775
C02740=1055.330,275.310,-99.935,172.683,36.067,156.776
C02741=1055.336,275.557,-99.964,172.686,36.070,156.777
C02742=1055.343,275.806,-99.995,172.688,36.074,156.778
C02743=1055.348,276.054,-100.025,172.691,36.077,156.778
C02744=1055.355,276.294,-100.055,172.694,36.081,156.779
C02745=1055.361,276.535,-100.085,172.697,36.084,156.780
C02746=1055.367,276.775,-100.115,172.700,36.088,156.781
C02747=1055.374,277.015,-100.144,172.702,36.092,156.781
C02748=1055.380,277.255,-100.173,172.705,36.095,156.782
C02749=1055.386,277.496,-100.202,172.708,36.099,156.783
C02750=1055.392,277.736,-100.233,172.711,36.102,156.784
C02751=1055.398,277.976,-100.262,172.713,36.106,156.784
C02752=1055.405,278.225,-100.293,172.716,36.109,156.785
C02753=1055.411,278.473,-100.323,172.719,36.113,156.786
C02754=1055.417,278.721,-100.354,172.722,36.116,156.787
C02755=1055.424,278.969,-100.385,172.725,36.120,156.787
C02756=1055.430,279.217,-100.415,172.728,36.123,156.788
C02757=1055.437,279.465,-100.446,172.730,36.127,156.789
C02758=1055.443,279.713,-100.477,172.734,36.130,156.790
C02759=1055.449,279.961,-100.507,172.736,36.134,156.790
C02760=1055.455,280.209,-100.538,172.740,36.138,156.791
C02761=1055.462,280.457,-100.569,172.742,36.141,156.792
C02762=1055.468,280.705,-100.600,172.745,36.145,156.793
C02763=1055.474,280.954,-100.631,172.748,36.148,156.793
C02764=1055.481,281.201,-100.662,172.750,36.152,156.794
C02765=1055.487,281.449,-100.692,172.754,36.155,156.795
C02766=1055.493,281.697,-100.723,172.756,36.160,156.796
C02767=1055.500,281.945,-100.754,172.760,36.163,156.797
C02768=1055.506,282.194,-100.785,172.762,36.167,156.797
C02769=1055.512,282.441,-100.816,172.765,36.170,156.798
C02770=1055.518,282.689,-100.847,172.768,36.174,156.799
C02771=1055.525,282.937,-100.878,172.771,36.178,156.800
C02772=1055.531,283.185,-100.908,172.774,36.181,156.800
C02773=1055.538,283.433,-100.940,172.777,36.185,156.801
C02774=1055.544,283.681,-100.971,172.780,36.188,156.802
C02775=1055.550,283.929,-101.002,172.783,36.192,156.803
C02776=1055.557,284.177,-101.033,172.786,36.196,156.804
C02777=1055.563,284.425,-101.064,172.789,36.199,156.804
C02778=1055.570,284.672,-101.095,172.792,36.203,156.805
C02779=1055.576,284.921,-101.126,172.795,36.206,156.806
C02780=1055.583,285.169,-101.157,172.798,36.210,156.807
C02781=1055.589,285.416,-101.188,172.801,36.214,156.807
C02782=1055.595,285.664,-101.219,172.804,36.217,156.808
C02783=1055.602,285.912,-101.250,172.806,36.221,156.809
C02784=1055.609,286.160,-101.282,172.810,36.224,156.810
C02785=1055.615,286.408,-101.312,172.812,36.228,156.810
C02786=1055.621,286.656,-101.343,172.816,36.231,156.811
C02787=1055.628,286.904,-101.375,172.819,36.236,156.812
C02788=1055.634,287.152,-101.406,172.822,36.239,156.813
C02789=1055.641,287.400,-101.437,172.825,36.243,156.814
C02790=1055.647,287.647,-101.468,172.827,36.246,156.814
C02791=1055.654,287.895,-101.500,172.831,36.250,156.815
C02792=1055.660,288.144,-101.532,172.833,36.254,156.816
C02793=1055.666,288.392,-101.562,172.837,36.257,156.817
C02794=1055.673,288.640,-101.594,172.840,36.261,156.818
C02795=1055.679,288.887,-101.625,172.843,36.265,156.818
C02796=1055.685,289.135,-101.657,172.846,36.268,156.819
C02797=1055.692,289.383,-101.688,172.849,36.272,156.820
C02798=1055.699,289.631,-101.720,172.852,36.276,156.821
C02799=1055.705,289.879,-101.751,172.855,36.279,156.822
C02800=1055.711,290.125,-101.783,172.858,36.283,156.822
C02801=1055.718,290.371,-101.813,172.861,36.286,156.823
C02802=1055.724,290.616,-101.845,172.864,36.290,156.824
C02803=1055.731,290.863,-101.876,172.867,36.294,156.825
C02804=1055.737,291.109,-101.907,172.870,36.297,156.825
C02805=1055.742,291.354,-101.939,172.873,36.301,156.826
C02806=1055.750,291.601,-101.970,172.877,36.305,156.827
C02807=1055.755,291.846,-102.001,172.879,36.308,156.828
C02808=1055.762,292.094,-102.033,172.882,36.312,156.829
C02809=1055.769,292.342,-102.064,172.886,36.316,156.830
C02810=1055.775,292.590,-102.096,172.888,36.320,156.830
C02811=1055.781,292.838,-102.127,172.892,36.324,156.831
C02812=1055.788,293.085,-102.159,172.894,36.327,156.832
C02813=1055.794,293.333,-102.191,172.898,36.331,156.833
C02814=1055.801,293.581,-102.223,172.901,36.335,156.834
C02815=1055.807,293.829,-102.255,172.904,36.338,156.834
C02816=1055.813,294.077,-102.286,172.907,36.342,156.835
C02817=1055.820,294.325,-102.318,172.911,36.346,156.836
C02818=1055.826,294.573,-102.351,172.913,36.349,156.837
C02819=1055.833,294.821,-102.382,172.917,36.353,156.838
C02820=1055.839,295.069,-102.414,172.920,36.357,156.838
C02821=1055.846,295.317,-102.445,172.922,36.360,156.839
C02822=1055.852,295.564,-102.478,172.926,36.364,156.840
C02823=1055.859,295.812,-102.510,172.929,36.368,156.841
C02824=1055.865,296.060,-102.542,172.932,36.372,156.842
C02825=1055.872,296.308,-102.574,172.935,36.375,156.842
C02826=1055.878,296.556,-102.606,172.939,36.379,156.843
C02827=1055.885,296.804,-102.637,172.941,36.383,156.844
C02828=1055.890,297.051,-102.670,172.945,36.387,156.845
C02829=1055.896,297.299,-102.702,172.948,36.390,156.846
C02830=1055.903,297.547,-102.734,172.951,36.394,156.847
C02831=1055.909,297.794,-102.766,172.954,36.399,156.848
C02832=1055.916,298.042,-102.799,172.958,36.402,156.848
C02833=1055.922,298.290,-102.831,172.960,36.406,156.849
C02834=1055.928,298.538,-102.863,172.964,36.410,156.850
C02835=1055.935,298.786,-102.895,172.967,36.414,156.851
C02836=1055.941,299.033,-102.928,172.971,36.418,156.852
C02837=1055.947,299.282,-102.960,172.973,36.421,156.853
C02838=1055.953,299.529,-102.992,172.977,36.425,156.853
C02839=1055.959,299.777,-103.024,172.980,36.429,156.854
C02840=1055.966,300.025,-103.056,172.983,36.433,156.855
C02841=1055.973,300.272,-103.089,172.986,36.437,156.856
C02842=1055.979,300.520,-103.121,172.990,36.441,156.857
C02843=1055.985,300.768,-103.154,172.993,36.444,156.858
C02844=1055.992,301.015,-103.186,172.996,36.448,156.858
C02845=1055.998,301.264,-103.218,172.999,36.452,156.859
C02846=1056.004,301.511,-103.251,173.003,36.456,156.860
C02847=1056.010,301.759,-103.284,173.006,36.460,156.861
C02848=1056.016,302.007,-103.316,173.009,36.463,156.862
C02849=1056.023,302.254,-103.348,173.012,36.467,156.863
C02850=1056.030,302.502,-103.381,173.016,36.471,156.864
C02851=1056.037,302.750,-103.414,173.019,36.475,156.864
C02852=1056.043,302.998,-103.446,173.022,36.479,156.865
C02853=1056.049,303.246,-103.478,173.025,36.483,156.866
C02854=1056.055,303.493,-103.511,173.029,36.487,156.867
C02855=1056.062,303.741,-103.544,173.032,36.491,156.868
C02856=1056.068,304.000,-103.578,173.036,36.495,156.869
C02857=1056.076,304.260,-103.612,173.038,36.499,156.870
C02858=1056.082,304.519,-103.646,173.042,36.503,156.870
C02859=1056.089,304.780,-103.680,173.045,36.507,156.871
C02860=1056.095,305.028,-103.713,173.049,36.511,156.872
C02861=1056.102,305.275,-103.745,173.052,36.515,156.873
C02862=1056.109,305.523,-103.778,173.056,36.518,156.874
C02863=1056.115,305.770,-103.811,173.059,36.522,156.875
C02864=1056.122,306.019,-103.844,173.062,36.526,156.876
C02865=1056.128,306.266,-103.877,173.065,36.530,156.877
C02866=1056.134,306.514,-103.909,173.069,36.534,156.877
C02867=1056.141,306.761,-103.942,173.072,36.538,156.878
C02868=1056.147,307.010,-103.975,173.076,36.542,156.879
C02869=1056.154,307.257,-104.007,173.079,36.545,156.880
C02870=1056.161,307.504,-104.040,173.082,36.549,156.881
C02871=1056.167,307.752,-104.073,173.085,36.553,156.882
C02872=1056.174,308.000,-104.107,173.089,36.557,156.883
C02873=1056.181,308.247,-104.139,173.092,36.561,156.883
C02874=1056.187,308.495,-104.172,173.096,36.565,156.884
C02875=1056.194,308.743,-104.205,173.100,36.569,156.885
C02876=1056.200,308.991,-104.238,173.103,36.573,156.886
C02877=1056.206,309.238,-104.271,173.106,36.576,156.887
C02878=1056.213,309.487,-104.304,173.109,36.581,156.888
C02879=1056.221,309.733,-104.337,173.113,36.585,156.889
C02880=1056.227,309.981,-104.369,173.116,36.589,156.890
C02881=1056.234,310.229,-104.403,173.120,36.593,156.890
C02882=1056.240,310.477,-104.435,173.123,36.596,156.891
C02883=1056.247,310.724,-104.469,173.127,36.600,156.892
C02884=1056.254,310.972,-104.502,173.130,36.604,156.893
C02885=1056.260,311.220,-104.535,173.134,36.608,156.894
C02886=1056.267,311.467,-104.568,173.136,36.612,156.895
C02887=1056.273,311.715,-104.601,173.140,36.616,156.896
C02888=1056.280,311.963,-104.634,173.143,36.620,156.897
C02889=1056.287,312.210,-104.668,173.147,36.624,156.897
C02890=1056.293,312.458,-104.700,173.150,36.628,156.898
C02891=1056.300,312.706,-104.734,173.154,36.632,156.899
C02892=1056.307,312.953,-104.767,173.158,36.636,156.900
C02893=1056.314,313.201,-104.800,173.161,36.639,156.901
C02894=1056.320,313.450,-104.833,173.165,36.643,156.902
C02895=1056.327,313.697,-104.867,173.168,36.647,156.903
C02896=1056.333,313.944,-104.901,173.172,36.651,156.904
C02897=1056.340,314.192,-104.934,173.174,36.656,156.905
C02898=1056.346,314.439,-104.968,173.178,36.660,156.906
C02899=1056.352,314.687,-105.001,173.181,36.664,156.906
C02900=1056.359,314.935,-105.034,173.185,36.668,156.907
C02901=1056.365,315.182,-105.069,173.189,36.672,156.908
C02902=1056.372,315.430,-105.102,173.192,36.676,156.909
C02903=1056.378,315.678,-105.136,173.196,36.680,156.910
C02904=1056.385,315.925,-105.170,173.199,36.684,156.911
C02905=1056.390,316.173,-105.203,173.203,36.688,156.912
C02906=1056.397,316.420,-105.236,173.206,36.692,156.913
C02907=1056.404,316.668,-105.271,173.210,36.696,156.914
C02908=1056.410,316.915,-105.304,173.214,36.700,156.915
C02909=1056.416,317.164,-105.338,173.217,36.705,156.916
C02910=1056.423,317.411,-105.371,173.221,36.709,156.917
C02911=1056.429,317.659,-105.406,173.223,36.713,156.918
C02912=1056.438,317.971,-105.449,173.228,36.718,156.919
C02913=1056.445,318.283,-105.491,173.233,36.723,156.920
C02914=1056.453,318.595,-105.534,173.238,36.728,156.921
C02915=1056.462,318.908,-105.576,173.241,36.734,156.922
C02916=1056.469,319.156,-105.610,173.245,36.738,156.923
C02917=1056.475,319.403,-105.644,173.249,36.742,156.924
C02918=1056.482,319.651,-105.678,173.252,36.746,156.925
C02919=1056.488,319.898,-105.712,173.256,36.751,156.926
C02920=1056.495,320.146,-105.746,173.259,36.755,156.927
C02921=1056.501,320.394,-105.780,173.263,36.759,156.928
C02922=1056.508,320.640,-105.814,173.266,36.763,156.929
C02923=1056.514,320.888,-105.848,173.270,36.767,156.930
C02924=1056.522,321.136,-105.882,173.274,36.771,156.931
C02925=1056.528,321.383,-105.916,173.277,36.775,156.932
C02926=1056.534,321.631,-105.950,173.282,36.780,156.933
C02927=1056.541,321.879,-105.984,173.286,36.784,156.934
C02928=1056.547,322.126,-106.018,173.289,36.788,156.935
C02929=1056.555,322.373,-106.053,173.293,36.792,156.936
C02930=1056.561,322.621,-106.087,173.296,36.796,156.936
C02931=1056.568,322.868,-106.121,173.300,36.800,156.937
C02932=1056.574,323.116,-106.155,173.304,36.805,156.938
C02933=1056.581,323.364,-106.190,173.307,36.809,156.939
C02934=1056.588,323.612,-106.223,173.311,36.813,156.940
C02935=1056.594,323.859,-106.257,173.314,36.817,156.941
C02936=1056.601,324.106,-106.292,173.318,36.821,156.942
C02937=1056.608,324.354,-106.326,173.322,36.826,156.943
C02938=1056.614,324.602,-106.361,173.325,36.830,156.944
C02939=1056.621,324.849,-106.394,173.329,36.834,156.945
C02940=1056.627,325.097,-106.429,173.332,36.839,156.946
C02941=1056.635,325.344,-106.463,173.336,36.843,156.947
C02942=1056.641,325.592,-106.498,173.341,36.847,156.948
C02943=1056.648,325.840,-106.533,173.344,36.851,156.949
C02944=1056.654,326.063,-106.564,173.347,36.855,156.950
C02945=1056.660,326.286,-106.595,173.351,36.859,156.951
C02946=1056.667,326.509,-106.626,173.354,36.862,156.952
C02947=1056.672,326.733,-106.657,173.358,36.866,156.952
C02948=1056.679,326.956,-106.688,173.361,36.870,156.953
C02949=1056.684,327.180,-106.719,173.365,36.874,156.954
C02950=1056.691,327.403,-106.750,173.367,36.878,156.955
C02951=1056.697,327.626,-106.782,173.371,36.882,156.956
C02952=1056.704,327.874,-106.815,173.375,36.886,156.957
C02953=1056.711,328.121,-106.851,173.378,36.890,156.958
C02954=1056.717,328.369,-106.885,173.383,36.895,156.959
C02955=1056.725,328.616,-106.920,173.386,36.899,156.960
C02956=1056.731,328.864,-106.954,173.390,36.903,156.961
C02957=1056.738,329.112,-106.989,173.394,36.907,156.962
C02958=1056.745,329.359,-107.023,173.397,36.912,156.963
C02959=1056.751,329.606,-107.058,173.401,36.916,156.964
C02960=1056.758,329.855,-107.092,173.406,36.920,156.965
C02961=1056.766,330.102,-107.127,173.409,36.925,156.966
C02962=1056.773,330.349,-107.162,173.413,36.929,156.967
C02963=1056.778,330.596,-107.196,173.417,36.933,156.968
C02964=1056.785,330.844,-107.231,173.420,36.938,156.969
C02965=1056.792,331.091,-107.266,173.424,36.942,156.970
C02966=1056.799,331.338,-107.302,173.429,36.946,156.971
C02967=1056.805,331.586,-107.337,173.432,36.951,156.972
C02968=1056.812,331.845,-107.374,173.436,36.955,156.973
C02969=1056.819,332.103,-107.410,173.440,36.960,156.974
C02970=1056.826,332.362,-107.447,173.444,36.965,156.975
C02971=1056.833,332.620,-107.483,173.448,36.970,156.976
C02972=1056.840,332.867,-107.518,173.452,36.974,156.977
C02973=1056.847,333.115,-107.553,173.457,36.979,156.978
C02974=1056.854,333.363,-107.588,173.460,36.983,156.979
C02975=1056.861,333.610,-107.624,173.464,36.988,156.980
C02976=1056.867,333.858,-107.659,173.468,36.992,156.981
C02977=1056.873,334.105,-107.694,173.471,36.996,156.982
C02978=1056.880,334.352,-107.730,173.476,37.001,156.984
C02979=1056.887,334.600,-107.765,173.480,37.005,156.985
C02980=1056.894,334.847,-107.800,173.483,37.010,156.986
C02981=1056.900,335.095,-107.835,173.487,37.014,156.987
C02982=1056.907,335.342,-107.870,173.492,37.019,156.988
C02983=1056.914,335.589,-107.905,173.495,37.023,156.989
C02984=1056.921,335.837,-107.940,173.499,37.028,156.990
C02985=1056.928,336.084,-107.977,173.503,37.032,156.991
C02986=1056.935,336.331,-108.012,173.508,37.037,156.992
C02987=1056.941,336.579,-108.047,173.511,37.041,156.993
C02988=1056.948,336.826,-108.083,173.515,37.046,156.994
C02989=1056.955,337.074,-108.118,173.519,37.050,156.995
C02990=1056.962,337.321,-108.154,173.524,37.055,156.996
C02991=1056.968,337.568,-108.189,173.527,37.060,156.997
C02992=1056.975,337.816,-108.225,173.531,37.064,156.998
C02993=1056.982,338.063,-108.261,173.536,37.069,156.999
C02994=1056.988,338.311,-108.296,173.539,37.073,157.000
C02995=1056.995,338.558,-108.332,173.543,37.078,157.002
C02996=1057.002,338.805,-108.367,173.547,37.083,157.003
C02997=1057.009,339.053,-108.403,173.552,37.087,157.004
C02998=1057.016,339.301,-108.439,173.555,37.092,157.005
C02999=1057.023,339.547,-108.474,173.559,37.096,157.006
C03000=1057.029,339.795,-108.510,173.564,37.101,157.007
C03001=1057.036,340.042,-108.546,173.568,37.106,157.008
C03002=1057.043,340.290,-108.582,173.571,37.110,157.009
C03003=1057.049,340.537,-108.618,173.576,37.116,157.010
C03004=1057.056,340.784,-108.653,173.580,37.120,157.011
C03005=1057.064,341.032,-108.689,173.584,37.125,157.013
C03006=1057.070,341.279,-108.725,173.588,37.130,157.014
C03007=1057.077,341.526,-108.761,173.592,37.134,157.015
C03008=1057.083,341.773,-108.797,173.596,37.139,157.016
C03009=1057.091,342.021,-108.833,173.601,37.144,157.017
C03010=1057.098,342.268,-108.869,173.604,37.148,157.018
C03011=1057.105,342.516,-108.906,173.609,37.153,157.019
C03012=1057.112,342.763,-108.941,173.613,37.158,157.020
C03013=1057.119,343.010,-108.977,173.617,37.162,157.021
C03014=1057.126,343.258,-109.013,173.621,37.167,157.023
C03015=1057.132,343.505,-109.049,173.625,37.172,157.024
C03016=1057.139,343.752,-109.085,173.629,37.177,157.025
C03017=1057.146,344.000,-109.122,173.634,37.181,157.026
C03018=1057.153,344.247,-109.158,173.638,37.186,157.027
C03019=1057.159,344.494,-109.194,173.642,37.191,157.028
C03020=1057.167,344.741,-109.230,173.646,37.196,157.029
C03021=1057.173,344.989,-109.266,173.650,37.201,157.031
C03022=1057.180,345.236,-109.303,173.655,37.205,157.032
C03023=1057.187,345.483,-109.339,173.658,37.210,157.033
C03024=1057.194,345.737,-109.377,173.663,37.215,157.034
C03025=1057.201,345.992,-109.414,173.667,37.220,157.035
C03026=1057.208,346.246,-109.452,173.672,37.225,157.036
C03027=1057.215,346.499,-109.488,173.676,37.230,157.038
C03028=1057.222,346.747,-109.525,173.681,37.235,157.039
C03029=1057.228,346.994,-109.561,173.684,37.240,157.040
C03030=1057.236,347.242,-109.598,173.689,37.245,157.041
C03031=1057.242,347.489,-109.634,173.693,37.250,157.042
C03032=1057.249,347.736,-109.671,173.698,37.254,157.043
C03033=1057.255,347.984,-109.707,173.702,37.259,157.044
C03034=1057.263,348.230,-109.744,173.706,37.264,157.046
C03035=1057.270,348.477,-109.781,173.710,37.270,157.047
C03036=1057.277,348.725,-109.818,173.715,37.275,157.048
C03037=1057.284,348.973,-109.854,173.719,37.280,157.049
C03038=1057.291,349.219,-109.891,173.723,37.284,157.050
C03039=1057.298,349.467,-109.928,173.728,37.289,157.052
C03040=1057.304,349.714,-109.964,173.731,37.294,157.053
C03041=1057.312,349.961,-110.000,173.736,37.299,157.054
C03042=1057.319,350.208,-110.038,173.741,37.304,157.055
C03043=1057.326,350.455,-110.074,173.745,37.309,157.056
C03044=1057.332,350.703,-110.111,173.750,37.314,157.058
C03045=1057.340,350.949,-110.148,173.754,37.319,157.059
C03046=1057.347,351.197,-110.185,173.759,37.324,157.060
C03047=1057.354,351.444,-110.222,173.762,37.329,157.061
C03048=1057.360,351.691,-110.259,173.767,37.334,157.062
C03049=1057.368,351.938,-110.296,173.771,37.339,157.064
C03050=1057.374,352.186,-110.333,173.776,37.344,157.065
C03051=1057.381,352.433,-110.370,173.780,37.350,157.066
C03052=1057.388,352.680,-110.407,173.785,37.355,157.067
C03053=1057.395,352.927,-110.444,173.789,37.360,157.069
C03054=1057.402,353.175,-110.481,173.794,37.365,157.070
C03055=1057.409,353.422,-110.518,173.797,37.370,157.071
C03056=1057.416,353.668,-110.556,173.802,37.375,157.072
C03057=1057.423,353.916,-110.592,173.807,37.380,157.073
C03058=1057.430,354.163,-110.630,173.811,37.385,157.075
C03059=1057.437,354.410,-110.667,173.816,37.390,157.076
C03060=1057.444,354.657,-110.705,173.820,37.396,157.077
C03061=1057.451,354.904,-110.741,173.825,37.401,157.078
C03062=1057.458,355.152,-110.779,173.830,37.406,157.080
C03063=1057.465,355.399,-110.816,173.834,37.411,157.081
C03064=1057.472,355.645,-110.854,173.838,37.416,157.082
C03065=1057.479,355.892,-110.891,173.842,37.422,157.084
C03066=1057.486,356.140,-110.928,173.847,37.427,157.085
C03067=1057.493,356.387,-110.965,173.852,37.432,157.086
C03068=1057.500,356.634,-111.003,173.856,37.438,157.087
C03069=1057.507,356.881,-111.040,173.861,37.442,157.089
C03070=1057.514,357.128,-111.078,173.866,37.448,157.090
C03071=1057.522,357.375,-111.115,173.870,37.453,157.091
C03072=1057.529,357.622,-111.153,173.875,37.459,157.092
C03073=1057.536,357.869,-111.190,173.880,37.464,157.094
C03074=1057.543,358.116,-111.228,173.884,37.469,157.095
C03075=1057.550,358.364,-111.266,173.889,37.474,157.096
C03076=1057.556,358.610,-111.303,173.894,37.480,157.098
C03077=1057.564,358.857,-111.341,173.898,37.485,157.099
C03078=1057.571,359.104,-111.378,173.902,37.490,157.100
C03079=1057.578,359.351,-111.416,173.907,37.496,157.101
C03080=1057.586,359.610,-111.456,173.911,37.501,157.103
C03081=1057.593,359.869,-111.496,173.916,37.507,157.104
C03082=1057.600,360.128,-111.535,173.922,37.513,157.106
C03083=1057.607,360.387,-111.575,173.927,37.518,157.107
C03084=1057.615,360.634,-111.612,173.932,37.524,157.108
C03085=1057.622,360.881,-111.650,173.937,37.529,157.110
C03086=1057.629,361.128,-111.689,173.940,37.534,157.111
C03087=1057.636,361.375,-111.726,173.945,37.540,157.112
C03088=1057.644,361.622,-111.764,173.950,37.545,157.114
C03089=1057.651,361.869,-111.802,173.954,37.551,157.115
C03090=1057.658,362.116,-111.841,173.959,37.556,157.116
C03091=1057.665,362.363,-111.878,173.964,37.562,157.118
C03092=1057.672,362.610,-111.917,173.969,37.567,157.119
C03093=1057.679,362.857,-111.955,173.973,37.573,157.120
C03094=1057.686,363.104,-111.993,173.978,37.578,157.122
C03095=1057.694,363.351,-112.031,173.983,37.584,157.123
C03096=1057.701,363.598,-112.070,173.988,37.589,157.124
C03097=1057.708,363.845,-112.107,173.993,37.595,157.126
C03098=1057.715,364.092,-112.146,173.997,37.600,157.127
C03099=1057.723,364.339,-112.184,174.002,37.606,157.128
C03100=1057.729,364.586,-112.222,174.007,37.611,157.130
C03101=1057.737,364.833,-112.261,174.013,37.618,157.131
C03102=1057.744,365.079,-112.299,174.017,37.623,157.133
C03103=1057.751,365.327,-112.337,174.022,37.629,157.134
C03104=1057.758,365.573,-112.376,174.027,37.635,157.136
C03105=1057.765,365.820,-112.414,174.032,37.640,157.137
C03106=1057.772,366.067,-112.453,174.037,37.646,157.138
C03107=1057.779,366.314,-112.492,174.041,37.651,157.140
C03108=1057.787,366.561,-112.530,174.046,37.657,157.141
C03109=1057.793,366.808,-112.568,174.051,37.663,157.142
C03110=1057.801,367.055,-112.607,174.056,37.669,157.144
C03111=1057.808,367.302,-112.646,174.061,37.674,157.145
C03112=1057.815,367.549,-112.685,174.066,37.680,157.147
C03113=1057.823,367.796,-112.723,174.071,37.686,157.148
C03114=1057.830,368.042,-112.762,174.075,37.692,157.150
C03115=1057.837,368.289,-112.800,174.080,37.697,157.151
C03116=1057.844,368.536,-112.839,174.086,37.703,157.153
C03117=1057.851,368.783,-112.878,174.091,37.709,157.154
C03118=1057.859,369.029,-112.917,174.096,37.715,157.155
C03119=1057.866,369.276,-112.956,174.101,37.720,157.157
C03120=1057.874,369.523,-112.994,174.106,37.726,157.158
C03121=1057.881,369.770,-113.033,174.111,37.732,157.160
C03122=1057.888,370.017,-113.072,174.116,37.738,157.161
C03123=1057.896,370.264,-113.111,174.121,37.744,157.163
C03124=1057.903,370.510,-113.150,174.125,37.750,157.164
C03125=1057.910,370.757,-113.189,174.130,37.755,157.165
C03126=1057.918,371.004,-113.228,174.136,37.761,157.167
C03127=1057.925,371.251,-113.267,174.141,37.767,157.168
C03128=1057.933,371.498,-113.307,174.146,37.773,157.170
C03129=1057.940,371.745,-113.345,174.151,37.779,157.171
C03130=1057.947,371.991,-113.384,174.156,37.785,157.173
C03131=1057.955,372.238,-113.424,174.161,37.791,157.174
C03132=1057.961,372.485,-113.462,174.166,37.797,157.176
C03133=1057.969,372.732,-113.502,174.172,37.803,157.177
C03134=1057.976,372.979,-113.541,174.177,37.809,157.179
C03135=1057.984,373.225,-113.580,174.182,37.815,157.180
C03136=1057.992,373.503,-113.624,174.187,37.822,157.182
C03137=1058.000,373.780,-113.669,174.194,37.828,157.184
C03138=1058.008,374.058,-113.713,174.199,37.836,157.186
C03139=1058.017,374.335,-113.758,174.205,37.843,157.187
C03140=1058.024,374.582,-113.797,174.211,37.849,157.189
C03141=1058.031,374.828,-113.837,174.216,37.855,157.190
C03142=1058.038,375.075,-113.876,174.221,37.861,157.192
C03143=1058.046,375.322,-113.916,174.226,37.867,157.194
C03144=1058.053,375.568,-113.955,174.231,37.873,157.195
C03145=1058.061,375.815,-113.995,174.237,37.879,157.197
C03146=1058.068,376.062,-114.035,174.242,37.886,157.198
C03147=1058.076,376.308,-114.075,174.247,37.892,157.200
C03148=1058.083,376.555,-114.114,174.252,37.898,157.201
C03149=1058.090,376.802,-114.154,174.257,37.904,157.203
C03150=1058.098,377.048,-114.194,174.263,37.910,157.204
C03151=1058.105,377.295,-114.233,174.268,37.917,157.206
C03152=1058.113,377.542,-114.273,174.274,37.923,157.208
C03153=1058.121,377.788,-114.313,174.279,37.929,157.209
C03154=1058.128,378.035,-114.353,174.285,37.935,157.211
C03155=1058.135,378.282,-114.393,174.290,37.942,157.212
C03156=1058.143,378.528,-114.433,174.295,37.948,157.214
C03157=1058.150,378.775,-114.472,174.300,37.954,157.216
C03158=1058.158,379.022,-114.512,174.306,37.961,157.217
C03159=1058.166,379.268,-114.552,174.311,37.967,157.219
C03160=1058.173,379.515,-114.592,174.317,37.973,157.220
C03161=1058.181,379.761,-114.632,174.323,37.980,157.222
C03162=1058.189,380.008,-114.672,174.328,37.986,157.224
C03163=1058.196,380.255,-114.712,174.333,37.992,157.225
C03164=1058.204,380.502,-114.752,174.338,37.999,157.227
C03165=1058.211,380.748,-114.793,174.344,38.005,157.229
C03166=1058.218,380.994,-114.833,174.350,38.012,157.230
C03167=1058.226,381.241,-114.873,174.355,38.018,157.232
C03168=1058.233,381.488,-114.914,174.361,38.025,157.234
C03169=1058.241,381.734,-114.954,174.366,38.031,157.235
C03170=1058.249,381.980,-114.994,174.372,38.038,157.237
C03171=1058.256,382.228,-115.035,174.377,38.045,157.239
C03172=1058.264,382.474,-115.075,174.383,38.051,157.240
C03173=1058.271,382.720,-115.116,174.389,38.058,157.242
C03174=1058.278,382.967,-115.156,174.394,38.064,157.244
C03175=1058.286,383.213,-115.197,174.399,38.071,157.245
C03176=1058.293,383.460,-115.238,174.406,38.078,157.247
C03177=1058.301,383.707,-115.278,174.411,38.084,157.249
C03178=1058.309,383.953,-115.319,174.416,38.091,157.250
C03179=1058.316,384.199,-115.360,174.422,38.098,157.252
C03180=1058.324,384.446,-115.400,174.428,38.104,157.254
C03181=1058.332,384.692,-115.440,174.434,38.111,157.256
C03182=1058.339,384.938,-115.481,174.439,38.118,157.257
C03183=1058.347,385.185,-115.522,174.444,38.125,157.259
C03184=1058.354,385.431,-115.563,174.451,38.131,157.261
C03185=1058.362,385.678,-115.604,174.456,38.138,157.263
C03186=1058.370,385.924,-115.644,174.462,38.145,157.264
C03187=1058.377,386.171,-115.686,174.468,38.151,157.266
C03188=1058.385,386.417,-115.726,174.473,38.158,157.268
C03189=1058.393,386.663,-115.767,174.479,38.165,157.270
C03190=1058.401,386.910,-115.808,174.485,38.172,157.271
C03191=1058.409,387.157,-115.850,174.491,38.178,157.273
C03192=1058.419,387.465,-115.900,174.498,38.187,157.275
C03193=1058.428,387.774,-115.952,174.505,38.196,157.278
C03194=1058.438,388.083,-116.003,174.512,38.205,157.280
C03195=1058.448,388.392,-116.055,174.520,38.213,157.282
C03196=1058.455,388.639,-116.096,174.526,38.220,157.284
C03197=1058.463,388.885,-116.137,174.532,38.227,157.286
C03198=1058.471,389.131,-116.177,174.538,38.234,157.288
C03199=1058.479,389.377,-116.219,174.544,38.241,157.289
C03200=1058.488,389.624,-116.260,174.550,38.248,157.291
C03201=1058.495,389.871,-116.302,174.555,38.255,157.293
C03202=1058.503,390.117,-116.344,174.562,38.262,157.295
C03203=1058.511,390.363,-116.384,174.567,38.269,157.297
C03204=1058.518,390.609,-116.426,174.574,38.276,157.299
C03205=1058.526,390.856,-116.468,174.579,38.283,157.300
C03206=1058.534,391.102,-116.509,174.586,38.291,157.302
C03207=1058.542,391.349,-116.550,174.591,38.298,157.304
C03208=1058.549,391.595,-116.592,174.598,38.305,157.306
C03209=1058.558,391.841,-116.634,174.604,38.312,157.308
C03210=1058.565,392.088,-116.675,174.610,38.319,157.310
C03211=1058.573,392.334,-116.717,174.616,38.327,157.312
C03212=1058.581,392.579,-116.759,174.622,38.333,157.314
C03213=1058.589,392.826,-116.800,174.628,38.341,157.316
C03214=1058.597,393.072,-116.842,174.635,38.348,157.317
C03215=1058.605,393.319,-116.884,174.640,38.355,157.319
C03216=1058.613,393.565,-116.926,174.647,38.363,157.321
C03217=1058.620,393.811,-116.968,174.652,38.370,157.323
C03218=1058.628,394.058,-117.011,174.659,38.378,157.325
C03219=1058.636,394.304,-117.053,174.665,38.385,157.327
C03220=1058.644,394.549,-117.094,174.671,38.392,157.329
C03221=1058.653,394.796,-117.136,174.677,38.400,157.331
C03222=1058.660,395.042,-117.178,174.684,38.407,157.333
C03223=1058.668,395.289,-117.220,174.690,38.415,157.335
C03224=1058.676,395.535,-117.262,174.696,38.422,157.337
C03225=1058.684,395.781,-117.305,174.703,38.430,157.339
C03226=1058.692,396.027,-117.347,174.708,38.437,157.341
C03227=1058.700,396.274,-117.389,174.715,38.444,157.343
C03228=1058.708,396.520,-117.431,174.722,38.452,157.345
C03229=1058.716,396.767,-117.473,174.728,38.460,157.347
C03230=1058.724,397.012,-117.516,174.734,38.467,157.349
C03231=1058.732,397.259,-117.558,174.741,38.475,157.351
C03232=1058.740,397.505,-117.600,174.747,38.482,157.353
C03233=1058.748,397.751,-117.643,174.753,38.490,157.355
C03234=1058.756,397.997,-117.685,174.760,38.498,157.357
C03235=1058.764,398.243,-117.727,174.766,38.506,157.359
C03236=1058.772,398.489,-117.770,174.773,38.513,157.361
C03237=1058.780,398.736,-117.813,174.780,38.521,157.363
C03238=1058.788,398.981,-117.855,174.785,38.529,157.365
C03239=1058.796,399.228,-117.898,174.792,38.537,157.367
C03240=1058.804,399.474,-117.941,174.799,38.544,157.369
C03241=1058.812,399.720,-117.983,174.806,38.552,157.371
C03242=1058.820,399.967,-118.026,174.811,38.560,157.374
C03243=1058.829,400.213,-118.069,174.818,38.568,157.376
C03244=1058.837,400.459,-118.112,174.825,38.576,157.378
C03245=1058.845,400.706,-118.155,174.832,38.584,157.380
C03246=1058.853,400.951,-118.198,174.838,38.591,157.382
C03247=1058.861,401.197,-118.241,174.845,38.599,157.384
C03248=1058.872,401.524,-118.298,174.853,38.610,157.387
C03249=1058.882,401.850,-118.354,174.863,38.620,157.390
C03250=1058.894,402.176,-118.411,174.871,38.631,157.393
C03251=1058.906,402.502,-118.469,174.881,38.641,157.395
C03252=1058.913,402.748,-118.512,174.887,38.650,157.398
C03253=1058.921,402.994,-118.555,174.893,38.658,157.400
C03254=1058.930,403.240,-118.598,174.900,38.666,157.402
C03255=1058.937,403.486,-118.642,174.907,38.674,157.404
C03256=1058.946,403.732,-118.685,174.914,38.682,157.406
C03257=1058.954,403.979,-118.729,174.921,38.690,157.409
C03258=1058.962,404.225,-118.772,174.928,38.698,157.411
C03259=1058.971,404.471,-118.815,174.935,38.707,157.413
C03260=1058.979,404.716,-118.859,174.941,38.715,157.415
C03261=1058.987,404.962,-118.902,174.948,38.723,157.418
C03262=1058.995,405.209,-118.946,174.955,38.732,157.420
C03263=1059.004,405.455,-118.989,174.962,38.740,157.422
C03264=1059.012,405.701,-119.033,174.969,38.748,157.424
C03265=1059.021,405.947,-119.076,174.976,38.757,157.427
C03266=1059.029,406.193,-119.121,174.983,38.765,157.429
C03267=1059.037,406.439,-119.164,174.990,38.773,157.431
C03268=1059.045,406.685,-119.208,174.997,38.782,157.433
C03269=1059.053,406.931,-119.252,175.004,38.790,157.436
C03270=1059.062,407.177,-119.296,175.011,38.799,157.438
C03271=1059.070,407.422,-119.340,175.018,38.807,157.440
C03272=1059.078,407.669,-119.383,175.025,38.816,157.443
C03273=1059.087,407.915,-119.428,175.033,38.824,157.445
C03274=1059.095,408.161,-119.472,175.040,38.833,157.447
C03275=1059.103,408.407,-119.516,175.047,38.842,157.450
C03276=1059.112,408.652,-119.559,175.054,38.850,157.452
C03277=1059.121,408.899,-119.604,175.061,38.859,157.455
C03278=1059.129,409.145,-119.648,175.069,38.867,157.457
C03279=1059.137,409.390,-119.692,175.076,38.876,157.459
C03280=1059.146,409.637,-119.737,175.083,38.885,157.462
C03281=1059.154,409.882,-119.781,175.091,38.894,157.464
C03282=1059.163,410.128,-119.825,175.098,38.902,157.466
C03283=1059.172,410.374,-119.870,175.105,38.911,157.469
C03284=1059.180,410.620,-119.914,175.112,38.920,157.471
C03285=1059.188,410.866,-119.959,175.120,38.929,157.474
C03286=1059.197,411.112,-120.002,175.128,38.938,157.476
C03287=1059.205,411.358,-120.047,175.135,38.946,157.479
C03288=1059.214,411.604,-120.091,175.142,38.955,157.481
C03289=1059.223,411.849,-120.136,175.149,38.964,157.484
C03290=1059.232,412.095,-120.181,175.158,38.973,157.486
C03291=1059.240,412.342,-120.225,175.165,38.982,157.489
C03292=1059.248,412.587,-120.270,175.172,38.991,157.491
C03293=1059.258,412.833,-120.314,175.180,39.000,157.493
C03294=1059.266,413.079,-120.359,175.188,39.009,157.496
C03295=1059.275,413.325,-120.404,175.195,39.018,157.499
C03296=1059.284,413.571,-120.449,175.202,39.027,157.501
C03297=1059.293,413.816,-120.493,175.211,39.036,157.504
C03298=1059.302,414.062,-120.538,175.218,39.045,157.506
C03299=1059.311,414.308,-120.583,175.226,39.054,157.509
C03300=1059.319,414.554,-120.628,175.234,39.063,157.511
C03301=1059.328,414.800,-120.673,175.241,39.073,157.514
C03302=1059.335,415.045,-120.719,175.249,39.082,157.516
C03303=1059.344,415.291,-120.764,175.257,39.091,157.519
C03304=1059.357,415.623,-120.825,175.267,39.104,157.523
C03305=1059.368,415.954,-120.886,175.278,39.116,157.526
C03306=1059.379,416.286,-120.947,175.289,39.129,157.530
C03307=1059.392,416.617,-121.008,175.299,39.142,157.533
C03308=1059.401,416.863,-121.054,175.307,39.151,157.536
C03309=1059.410,417.109,-121.099,175.315,39.161,157.539
C03310=1059.418,417.354,-121.144,175.324,39.170,157.541
C03311=1059.427,417.600,-121.190,175.331,39.180,157.544
C03312=1059.436,417.846,-121.235,175.340,39.189,157.547
C03313=1059.445,418.091,-121.281,175.347,39.199,157.549
C03314=1059.454,418.337,-121.327,175.356,39.209,157.552
C03315=1059.462,418.583,-121.373,175.364,39.218,157.555
C03316=1059.471,418.829,-121.418,175.372,39.228,157.557
C03317=1059.480,419.074,-121.464,175.380,39.238,157.560
C03318=1059.490,419.320,-121.510,175.388,39.247,157.563
C03319=1059.499,419.565,-121.555,175.397,39.257,157.566
C03320=1059.508,419.811,-121.601,175.405,39.267,157.568
C03321=1059.517,420.057,-121.647,175.413,39.276,157.571
C03322=1059.526,420.302,-121.693,175.421,39.286,157.574
C03323=1059.534,420.548,-121.739,175.430,39.296,157.577
C03324=1059.544,420.793,-121.785,175.438,39.306,157.580
C03325=1059.552,421.039,-121.832,175.447,39.316,157.583
C03326=1059.561,421.284,-121.877,175.455,39.326,157.585
C03327=1059.570,421.530,-121.924,175.463,39.336,157.588
C03328=1059.580,421.776,-121.970,175.472,39.346,157.591
C03329=1059.589,422.021,-122.016,175.481,39.356,157.594
C03330=1059.598,422.267,-122.063,175.489,39.366,157.597
C03331=1059.607,422.512,-122.109,175.498,39.376,157.600
C03332=1059.615,422.757,-122.156,175.506,39.387,157.603
C03333=1059.625,423.003,-122.203,175.515,39.396,157.605
C03334=1059.634,423.249,-122.249,175.523,39.407,157.608
C03335=1059.643,423.494,-122.295,175.532,39.417,157.611
C03336=1059.652,423.739,-122.342,175.541,39.427,157.614
C03337=1059.662,423.985,-122.389,175.550,39.437,157.617
C03338=1059.671,424.231,-122.435,175.559,39.448,157.620
C03339=1059.680,424.475,-122.482,175.567,39.458,157.623
C03340=1059.690,424.721,-122.529,175.576,39.468,157.626
C03341=1059.698,424.967,-122.575,175.585,39.479,157.629
C03342=1059.708,425.211,-122.622,175.593,39.489,157.632
C03343=1059.717,425.458,-122.669,175.602,39.499,157.635
C03344=1059.726,425.703,-122.716,175.611,39.510,157.638
C03345=1059.736,425.948,-122.763,175.620,39.520,157.641
C03346=1059.745,426.194,-122.810,175.629,39.531,157.644
C03347=1059.754,426.439,-122.857,175.638,39.542,157.648
C03348=1059.764,426.684,-122.905,175.647,39.552,157.651
C03349=1059.773,426.930,-122.951,175.656,39.563,157.654
C03350=1059.782,427.176,-122.999,175.666,39.574,157.657
C03351=1059.792,427.420,-123.046,175.675,39.584,157.660
C03352=1059.802,427.666,-123.094,175.684,39.595,157.663
C03353=1059.810,427.911,-123.140,175.694,39.606,157.666
C03354=1059.820,428.157,-123.188,175.703,39.617,157.669
C03355=1059.830,428.402,-123.235,175.712,39.628,157.673
C03356=1059.839,428.647,-123.283,175.721,39.638,157.676
C03357=1059.848,428.893,-123.331,175.731,39.649,157.679
C03358=1059.858,429.138,-123.378,175.740,39.660,157.682
C03359=1059.867,429.382,-123.426,175.750,39.671,157.685
C03360=1059.878,429.651,-123.478,175.760,39.684,157.689
C03361=1059.888,429.919,-123.530,175.771,39.695,157.692
C03362=1059.898,430.188,-123.583,175.781,39.707,157.696
C03363=1059.909,430.457,-123.635,175.792,39.720,157.700
C03364=1059.919,430.703,-123.683,175.801,39.731,157.703
C03365=1059.928,430.947,-123.731,175.810,39.742,157.706
C03366=1059.937,431.193,-123.779,175.820,39.754,157.710
C03367=1059.947,431.438,-123.828,175.830,39.765,157.713
C03368=1059.957,431.683,-123.876,175.839,39.776,157.716
C03369=1059.966,431.928,-123.924,175.850,39.788,157.720
C03370=1059.976,432.173,-123.973,175.859,39.799,157.723
C03371=1059.985,432.419,-124.020,175.869,39.810,157.727
C03372=1059.996,432.663,-124.068,175.879,39.821,157.730
C03373=1060.005,432.909,-124.117,175.888,39.833,157.733
C03374=1060.015,433.154,-124.166,175.899,39.845,157.737
C03375=1060.025,433.399,-124.214,175.908,39.856,157.740
C03376=1060.034,433.644,-124.263,175.919,39.868,157.744
C03377=1060.044,433.889,-124.312,175.928,39.880,157.747
C03378=1060.054,434.134,-124.360,175.939,39.891,157.751
C03379=1060.064,434.379,-124.409,175.949,39.903,157.754
C03380=1060.073,434.624,-124.457,175.959,39.914,157.758
C03381=1060.083,434.869,-124.506,175.970,39.926,157.761
C03382=1060.093,435.114,-124.554,175.979,39.938,157.765
C03383=1060.104,435.359,-124.604,175.990,39.949,157.768
C03384=1060.113,435.604,-124.652,176.000,39.962,157.772
C03385=1060.123,435.849,-124.701,176.011,39.974,157.775
C03386=1060.133,436.093,-124.750,176.021,39.985,157.779
C03387=1060.143,436.339,-124.799,176.032,39.997,157.783
C03388=1060.154,436.583,-124.848,176.042,40.009,157.786
C03389=1060.163,436.828,-124.897,176.053,40.021,157.790
C03390=1060.174,437.073,-124.946,176.063,40.033,157.794
C03391=1060.184,437.318,-124.995,176.073,40.045,157.797
C03392=1060.194,437.563,-125.044,176.084,40.057,157.801
C03393=1060.204,437.808,-125.094,176.095,40.070,157.805
C03394=1060.214,438.052,-125.144,176.106,40.082,157.808
C03395=1060.224,438.297,-125.193,176.117,40.094,157.812
C03396=1060.234,438.542,-125.243,176.128,40.106,157.816
C03397=1060.244,438.787,-125.293,176.138,40.119,157.820
C03398=1060.254,439.031,-125.342,176.149,40.131,157.823
C03399=1060.265,439.276,-125.391,176.160,40.144,157.827
C03400=1060.274,439.521,-125.441,176.171,40.156,157.831
C03401=1060.285,439.766,-125.491,176.182,40.169,157.835
C03402=1060.295,440.011,-125.541,176.193,40.181,157.839
C03403=1060.305,440.256,-125.590,176.204,40.194,157.843
C03404=1060.316,440.500,-125.641,176.216,40.207,157.847
C03405=1060.325,440.745,-125.691,176.227,40.219,157.850
C03406=1060.336,440.989,-125.741,176.238,40.232,157.854
C03407=1060.346,441.234,-125.791,176.249,40.245,157.858
C03408=1060.357,441.479,-125.841,176.260,40.257,157.862
C03409=1060.367,441.724,-125.891,176.271,40.270,157.866
C03410=1060.378,441.968,-125.942,176.283,40.283,157.870
C03411=1060.389,442.212,-125.992,176.295,40.296,157.874
C03412=1060.399,442.458,-126.042,176.306,40.309,157.878
C03413=1060.410,442.702,-126.092,176.317,40.322,157.882
C03414=1060.420,442.947,-126.143,176.330,40.335,157.886
C03415=1060.430,443.192,-126.194,176.341,40.348,157.890
C03416=1060.444,443.526,-126.263,176.357,40.366,157.896
C03417=1060.461,443.910,-126.342,176.375,40.387,157.903
C03418=1060.478,444.293,-126.422,176.394,40.408,157.909
C03419=1060.494,444.676,-126.502,176.413,40.428,157.916
C03420=1060.510,445.060,-126.582,176.432,40.450,157.922
C03421=1060.522,445.304,-126.633,176.443,40.463,157.926
C03422=1060.532,445.548,-126.684,176.456,40.477,157.931
C03423=1060.543,445.792,-126.736,176.467,40.490,157.935
C03424=1060.554,446.038,-126.786,176.480,40.504,157.939
C03425=1060.565,446.282,-126.838,176.492,40.518,157.944
C03426=1060.575,446.526,-126.889,176.504,40.531,157.948
C03427=1060.586,446.770,-126.940,176.517,40.545,157.952
C03428=1060.597,447.015,-126.992,176.530,40.558,157.957
C03429=1060.608,447.257,-127.043,176.541,40.572,157.961
C03430=1060.620,447.501,-127.094,176.554,40.586,157.965
C03431=1060.632,447.745,-127.143,176.567,40.599,157.970
C03432=1060.646,447.990,-127.193,176.579,40.612,157.974
C03433=1060.661,448.234,-127.242,176.592,40.625,157.978
C03434=1060.676,448.477,-127.290,176.605,40.638,157.982
C03435=1060.692,448.723,-127.338,176.618,40.650,157.986
C03436=1060.709,448.968,-127.385,176.631,40.662,157.990
C03437=1060.728,449.212,-127.432,176.644,40.674,157.994
C03438=1060.746,449.457,-127.477,176.657,40.685,157.998
C03439=1060.765,449.702,-127.523,176.671,40.697,158.002
C03440=1060.787,449.948,-127.567,176.684,40.708,158.005
C03441=1060.455,449.960,-127.844,176.679,40.822,158.037
C03442=1060.434,449.714,-127.799,176.665,40.811,158.033
C03443=1060.414,449.468,-127.755,176.651,40.800,158.029
C03444=1060.395,449.223,-127.709,176.638,40.788,158.025
C03445=1060.377,448.978,-127.663,176.625,40.776,158.021
C03446=1060.360,448.733,-127.615,176.612,40.764,158.017
C03447=1060.343,448.489,-127.568,176.599,40.752,158.013
C03448=1060.328,448.244,-127.519,176.586,40.740,158.009
C03449=1060.313,448.000,-127.471,176.573,40.727,158.005
C03450=1060.299,447.756,-127.422,176.560,40.714,158.001
C03451=1060.287,447.512,-127.371,176.548,40.700,157.997
C03452=1060.275,447.269,-127.321,176.535,40.687,157.992
C03453=1060.264,447.026,-127.269,176.522,40.674,157.988
C03454=1060.252,446.782,-127.218,176.510,40.660,157.984
C03455=1060.242,446.537,-127.167,176.498,40.646,157.979
C03456=1060.231,446.293,-127.115,176.485,40.633,157.975
C03457=1060.219,446.048,-127.064,176.473,40.619,157.971
C03458=1060.209,445.803,-127.013,176.461,40.605,157.966
C03459=1060.199,445.559,-126.961,176.448,40.592,157.962
C03460=1060.187,445.316,-126.910,176.436,40.578,157.958
C03461=1060.177,445.071,-126.860,176.424,40.565,157.953
C03462=1060.161,444.707,-126.783,176.406,40.545,157.947
C03463=1060.145,444.343,-126.707,176.388,40.526,157.941
C03464=1060.129,443.978,-126.632,176.371,40.506,157.935
C03465=1060.113,443.615,-126.556,176.353,40.486,157.929
C03466=1060.103,443.370,-126.505,176.340,40.473,157.924
C03467=1060.092,443.125,-126.455,176.329,40.460,157.920
C03468=1060.082,442.881,-126.404,176.318,40.447,157.916
C03469=1060.071,442.636,-126.354,176.305,40.434,157.912
C03470=1060.061,442.391,-126.303,176.294,40.421,157.908
C03471=1060.050,442.147,-126.253,176.283,40.408,157.904
C03472=1060.040,441.902,-126.203,176.270,40.395,157.900
C03473=1060.029,441.658,-126.152,176.259,40.382,157.896
C03474=1060.019,441.413,-126.102,176.248,40.370,157.892
C03475=1060.008,441.168,-126.052,176.237,40.357,157.888
C03476=1059.998,440.924,-126.001,176.226,40.344,157.884
C03477=1059.988,440.679,-125.952,176.213,40.332,157.880
C03478=1059.977,440.435,-125.901,176.202,40.319,157.876
C03479=1059.967,440.189,-125.851,176.191,40.307,157.872
C03480=1059.957,439.945,-125.802,176.180,40.294,157.869
C03481=1059.947,439.700,-125.751,176.169,40.281,157.865
C03482=1059.936,439.455,-125.701,176.158,40.269,157.861
C03483=1059.926,439.211,-125.652,176.147,40.257,157.857
C03484=1059.915,438.966,-125.602,176.136,40.244,157.853
C03485=1059.906,438.721,-125.553,176.125,40.232,157.849
C03486=1059.895,438.476,-125.503,176.114,40.219,157.846
C03487=1059.885,438.232,-125.454,176.103,40.207,157.842
C03488=1059.875,437.986,-125.404,176.092,40.195,157.838
C03489=1059.865,437.742,-125.354,176.081,40.183,157.834
C03490=1059.855,437.497,-125.305,176.071,40.171,157.831
C03491=1059.845,437.252,-125.256,176.060,40.158,157.827
C03492=1059.834,437.007,-125.207,176.050,40.146,157.823
C03493=1059.825,436.762,-125.157,176.039,40.134,157.820
C03494=1059.811,436.439,-125.093,176.025,40.119,157.815
C03495=1059.798,436.114,-125.028,176.011,40.103,157.810
C03496=1059.784,435.791,-124.963,175.997,40.087,157.805
C03497=1059.771,435.467,-124.898,175.983,40.072,157.801
C03498=1059.761,435.222,-124.849,175.973,40.060,157.797
C03499=1059.752,434.977,-124.801,175.963,40.048,157.793
C03500=1059.742,434.732,-124.751,175.952,40.037,157.790
C03501=1059.732,434.487,-124.702,175.942,40.024,157.786
C03502=1059.722,434.242,-124.654,175.932,40.013,157.783
C03503=1059.712,433.997,-124.605,175.921,40.001,157.779
C03504=1059.703,433.752,-124.557,175.912,39.990,157.776
C03505=1059.693,433.507,-124.508,175.901,39.978,157.772
C03506=1059.683,433.262,-124.460,175.891,39.967,157.769
C03507=1059.673,433.017,-124.411,175.881,39.956,157.765
C03508=1059.664,432.772,-124.362,175.871,39.944,157.762
C03509=1059.654,432.527,-124.314,175.861,39.932,157.758
C03510=1059.644,432.282,-124.265,175.852,39.921,157.755
C03511=1059.635,432.037,-124.218,175.841,39.910,157.752
C03512=1059.625,431.792,-124.169,175.832,39.898,157.748
C03513=1059.615,431.547,-124.121,175.821,39.887,157.745
C03514=1059.606,431.301,-124.073,175.812,39.876,157.742
C03515=1059.596,431.056,-124.024,175.802,39.864,157.738
C03516=1059.586,430.811,-123.976,175.792,39.853,157.735
C03517=1059.577,430.566,-123.929,175.783,39.842,157.732
C03518=1059.565,430.291,-123.875,175.772,39.830,157.728
C03519=1059.555,430.015,-123.821,175.761,39.817,157.724
C03520=1059.544,429.740,-123.767,175.751,39.805,157.721
C03521=1059.533,429.464,-123.713,175.740,39.792,157.717
C03522=1059.524,429.219,-123.666,175.730,39.782,157.714
C03523=1059.514,428.974,-123.618,175.720,39.771,157.710
C03524=1059.505,428.728,-123.570,175.711,39.760,157.707
C03525=1059.495,428.483,-123.523,175.702,39.749,157.704
C03526=1059.486,428.238,-123.475,175.693,39.738,157.701
C03527=1059.476,427.992,-123.428,175.683,39.728,157.698
C03528=1059.467,427.748,-123.381,175.674,39.717,157.695
C03529=1059.457,427.502,-123.333,175.664,39.706,157.691
C03530=1059.448,427.256,-123.285,175.655,39.695,157.688
C03531=1059.438,427.012,-123.238,175.646,39.685,157.685
C03532=1059.429,426.766,-123.191,175.637,39.674,157.682
C03533=1059.420,426.521,-123.144,175.628,39.663,157.679
C03534=1059.410,426.275,-123.097,175.619,39.653,157.676
C03535=1059.402,426.030,-123.050,175.610,39.642,157.673
C03536=1059.391,425.785,-123.003,175.601,39.632,157.670
C03537=1059.383,425.539,-122.956,175.592,39.621,157.667
C03538=1059.373,425.294,-122.909,175.583,39.611,157.664
C03539=1059.364,425.048,-122.862,175.574,39.600,157.660
C03540=1059.354,424.803,-122.815,175.565,39.590,157.658
C03541=1059.345,424.558,-122.768,175.556,39.580,157.655
C03542=1059.336,424.312,-122.721,175.547,39.570,157.652
C03543=1059.327,424.066,-122.675,175.538,39.559,157.649
C03544=1059.317,423.822,-122.628,175.529,39.549,157.646
C03545=1059.308,423.576,-122.581,175.520,39.539,157.643
C03546=1059.299,423.330,-122.535,175.511,39.529,157.640
C03547=1059.290,423.085,-122.489,175.503,39.518,157.637
C03548=1059.281,422.839,-122.441,175.494,39.508,157.634
C03549=1059.271,422.594,-122.395,175.486,39.498,157.631
C03550=1059.263,422.348,-122.349,175.477,39.488,157.628
C03551=1059.253,422.103,-122.302,175.468,39.478,157.625
C03552=1059.244,421.858,-122.256,175.459,39.468,157.622
C03553=1059.235,421.611,-122.209,175.451,39.458,157.619
C03554=1059.226,421.366,-122.163,175.443,39.448,157.616
C03555=1059.217,421.121,-122.116,175.434,39.438,157.614
C03556=1059.208,420.875,-122.071,175.425,39.429,157.611
C03557=1059.199,420.630,-122.025,175.418,39.419,157.608
C03558=1059.190,420.384,-121.978,175.409,39.408,157.605
C03559=1059.181,420.138,-121.933,175.400,39.399,157.602
C03560=1059.172,419.893,-121.887,175.393,39.389,157.599
C03561=1059.163,419.647,-121.841,175.384,39.379,157.597
C03562=1059.154,419.402,-121.795,175.375,39.370,157.594
C03563=1059.146,419.156,-121.749,175.368,39.360,157.591
C03564=1059.136,418.911,-121.703,175.359,39.350,157.588
C03565=1059.127,418.665,-121.657,175.350,39.341,157.586
C03566=1059.118,418.419,-121.612,175.343,39.331,157.583
C03567=1059.109,418.174,-121.566,175.334,39.322,157.580
C03568=1059.100,417.928,-121.520,175.327,39.312,157.578
C03569=1059.091,417.682,-121.475,175.318,39.303,157.575
C03570=1059.082,417.436,-121.430,175.309,39.293,157.572
C03571=1059.073,417.191,-121.384,175.302,39.283,157.569
C03572=1059.065,416.945,-121.337,175.293,39.274,157.567
C03573=1059.056,416.699,-121.292,175.286,39.265,157.564
C03574=1059.044,416.366,-121.231,175.275,39.252,157.561
C03575=1059.032,416.032,-121.169,175.264,39.239,157.557
C03576=1059.020,415.699,-121.108,175.254,39.226,157.553
C03577=1059.008,415.365,-121.047,175.242,39.214,157.550
C03578=1058.999,415.119,-121.001,175.235,39.205,157.547
C03579=1058.991,414.874,-120.956,175.227,39.195,157.545
C03580=1058.982,414.628,-120.911,175.219,39.186,157.542
C03581=1058.973,414.382,-120.866,175.212,39.177,157.539
C03582=1058.965,414.137,-120.821,175.203,39.168,157.537
C03583=1058.956,413.891,-120.776,175.196,39.159,157.534
C03584=1058.947,413.645,-120.731,175.188,39.149,157.532
C03585=1058.939,413.399,-120.686,175.180,39.141,157.529
C03586=1058.930,413.153,-120.641,175.173,39.131,157.527
C03587=1058.920,412.907,-120.596,175.165,39.122,157.524
C03588=1058.912,412.662,-120.552,175.157,39.114,157.522
C03589=1058.903,412.416,-120.507,175.150,39.105,157.519
C03590=1058.894,412.170,-120.463,175.142,39.096,157.517
C03591=1058.886,411.924,-120.418,175.135,39.087,157.514
C03592=1058.878,411.678,-120.374,175.127,39.078,157.512
C03593=1058.869,411.432,-120.328,175.120,39.069,157.509
C03594=1058.860,411.187,-120.285,175.112,39.060,157.507
C03595=1058.851,410.941,-120.240,175.105,39.051,157.504
C03596=1058.843,410.695,-120.196,175.097,39.043,157.502
C03597=1058.834,410.449,-120.152,175.089,39.034,157.499
C03598=1058.826,410.203,-120.107,175.082,39.025,157.497
C03599=1058.817,409.956,-120.062,175.075,39.016,157.495
C03600=1058.809,409.711,-120.018,175.068,39.007,157.492
C03601=1058.800,409.465,-119.974,175.061,38.999,157.490
C03602=1058.791,409.219,-119.930,175.053,38.990,157.487
C03603=1058.783,408.973,-119.885,175.045,38.982,157.485
C03604=1058.775,408.728,-119.842,175.038,38.973,157.483
C03605=1058.766,408.481,-119.797,175.031,38.965,157.480
C03606=1058.758,408.235,-119.753,175.024,38.956,157.478
C03607=1058.749,407.990,-119.709,175.017,38.947,157.476
C03608=1058.741,407.744,-119.665,175.010,38.939,157.473
C03609=1058.732,407.498,-119.621,175.002,38.930,157.471
C03610=1058.724,407.252,-119.577,174.995,38.922,157.469
C03611=1058.716,407.005,-119.533,174.988,38.914,157.466
C03612=1058.707,406.760,-119.489,174.981,38.905,157.464
C03613=1058.699,406.514,-119.445,174.974,38.897,157.462
C03614=1058.691,406.268,-119.401,174.967,38.888,157.459
C03615=1058.682,406.022,-119.357,174.960,38.880,157.457
C03616=1058.674,405.775,-119.314,174.953,38.872,157.455
C03617=1058.665,405.530,-119.270,174.946,38.863,157.453
C03618=1058.658,405.284,-119.226,174.939,38.855,157.450
C03619=1058.649,405.038,-119.183,174.932,38.847,157.448
C03620=1058.641,404.792,-119.139,174.925,38.838,157.446
C03621=1058.633,404.546,-119.096,174.918,38.830,157.443
C03622=1058.625,404.299,-119.052,174.911,38.822,157.441
C03623=1058.616,404.053,-119.009,174.904,38.814,157.439
C03624=1058.608,403.808,-118.966,174.898,38.806,157.437
